	Mission^.XPick			:= WorkArea^[Mission^.PPick].X;// + (Layer^[WorkArea^[Mission^.PPick].Layer].X / 2); (* valorizzo la quota X di prelievo  *)
	Mission^.YPick			:= WorkArea^[Mission^.PPick].Y + (Layer^[WorkPickPointState^[Mission^.PPick].Code].YDim / 2); (* valorizzo la quota Y di prelievo *)
	Mission^.ZPick			:= WorkArea^[Mission^.PPick].Z; (* in questo modo LA LENTA va sempre fino a zero...mi fermo al raggiungimento dell'intervento dei tastatori *)
ELSE
	Errore.Code := ErrWAM_TipologiaMagazzinoFaldaNONRiconosciuta; (*Errore, Nell'impianto è stata impostata una tipologia di magazzino falde non prevista!!!*)
	RETURN;//EXIT;
END_IF
//IF WorkAreaState^[cwa].P = 0 THEN (* Se devo depositare la falda su una CASSA/CAVALLETTO *)
//(*******************************************************************************************************************************)	
//(********************************************* DEPOSITO FALDA SU CASSA/CAVALLETTO **********************************************)
//(*******************************************************************************************************************************)
TFWAM_CreaMissione_DepFaldaSuPallet(NPosInLavoro			:= Mission^.PPlace, //Numero Postazione di depositio
									Angolo_Destinazione 	:= Forming^[WorkAreaState^[Mission^.PPlace].F].PElement[WorkAreaState^[Mission^.PPlace].P].J, //Angolo di deposito dell'elemento
									PosizioneAttuale_X      := ModuleAX_X^.Ax^.Status.ActPosition, //Posizione attuale asse X
									TipologiaTraiettoria    := Forming^[WorkAreaState^[cwa].F].PElement[WorkAreaState^[cwa].P].Trajectory,
									
									Quota_PostX				:= WorkArea^[Mission^.PPlace].X, //Quota X Postazione
									Quota_PostY				:= WorkArea^[Mission^.PPlace].Y, //Quota Y Postazione
									Quota_PostZ				:= WorkArea^[Mission^.PPlace].Z, //Quota Z Postazione
									Quota_PostJ				:= WorkArea^[Mission^.PPlace].Rx, //Quota J Postazione
									
									Offset_Postazione_X 	:= WorkAreaOffset^[Mission^.PPlace].X, //Offset X Postazione
									Offset_Postazione_Y 	:= WorkAreaOffset^[Mission^.PPlace].Y, //Offset Y Postazione
									Offset_Postazione_Z 	:= WorkAreaOffset^[Mission^.PPlace].Z, //Offset Z Postazione
									Offset_Postazione_J 	:= WorkAreaOffset^[Mission^.PPlace].Rx, //Offset J Postazione
									
									Pallet_DimX				:= Forming^[WorkAreaState^[Mission^.PPlace].F].Pallet.XDim, //Dimensione X Pallet
									Pallet_DimY				:= Forming^[WorkAreaState^[Mission^.PPlace].F].Pallet.YDim, //Dimensione Y Pallet
									Pallet_DimZ				:= Forming^[WorkAreaState^[Mission^.PPlace].F].Pallet.ZDim, //Dimensione Z Pallet
									
									Offset_Pallet_X_0		:= Forming^[WorkAreaState^[Mission^.PPlace].F].Pallet.OFSDE_X0, //Offset X Pallet o Casse
									Offset_Pallet_Y_0		:= Forming^[WorkAreaState^[Mission^.PPlace].F].Pallet.OFSDE_Y0, //Offset Y Pallet o Casse 
									Offset_Pallet_Z_0		:= Forming^[WorkAreaState^[Mission^.PPlace].F].Pallet.OFSDE_Z0, //Offset Z Pallet o Casse + è grande + il deposito si distanzia dal supporto
									Offset_Pallet_J_0		:= Forming^[WorkAreaState^[Mission^.PPlace].F].Pallet.OFSDE_J0, //Offset J Pallet o Casse + è grande + la lastra sarà inclinata verso l'angolo crescente
									
									Offset_Pallet_X_90		:= Forming^[WorkAreaState^[Mission^.PPlace].F].Pallet.OFSDE_X90, //Offset X Pallet lato 0-90 
									Offset_Pallet_Y_90		:= Forming^[WorkAreaState^[Mission^.PPlace].F].Pallet.OFSDE_Y90, //Offset Y Pallet lato 0-90 + è grande + il deposito si distanzia dal supporto
									Offset_Pallet_Z_90		:= Forming^[WorkAreaState^[Mission^.PPlace].F].Pallet.OFSDE_Z90, //Offset Z Pallet lato 0-90 + è grande + il deposito si distanzia dal supporto
									Offset_Pallet_J_90		:= Forming^[WorkAreaState^[Mission^.PPlace].F].Pallet.OFSDE_J90, //Offset J Pallet lato 0-90 + è grande + la lastra sarà inclinata in fase di deposito
									
									Offset_Pallet_X_180		:= Forming^[WorkAreaState^[Mission^.PPlace].F].Pallet.OFSDE_X180, //Offset X Pallet lato 90-180
									Offset_Pallet_Y_180		:= Forming^[WorkAreaState^[Mission^.PPlace].F].Pallet.OFSDE_Y180, //Offset Y Pallet lato 90-180 + è grande + il deposito si distanzia dal supporto
									Offset_Pallet_Z_180		:= Forming^[WorkAreaState^[Mission^.PPlace].F].Pallet.OFSDE_Z180, //Offset Z Pallet lato 90-180 + è grande + il deposito si distanzia dal supporto
									Offset_Pallet_J_180		:= Forming^[WorkAreaState^[Mission^.PPlace].F].Pallet.OFSDE_J180, //Offset J Pallet lato 90-180 + è grande + la lastra sarà inclinata in fase di deposito
									
									Quota_FormaturaX 		:= Forming^[WorkAreaState^[Mission^.PPlace].F].PElement[WorkAreaState^[Mission^.PPlace].P].X, //Quota Deposito X da Formatura
									Quota_FormaturaY 		:= Forming^[WorkAreaState^[Mission^.PPlace].F].PElement[WorkAreaState^[Mission^.PPlace].P].Y, //Quota Deposito Y da Formatura
									Quota_FormaturaZ 		:= Forming^[WorkAreaState^[Mission^.PPlace].F].PElement[WorkAreaState^[Mission^.PPlace].P].Z, //Quota Deposito Z da Formatura
									Quota_FormaturaJ 		:= Forming^[WorkAreaState^[Mission^.PPlace].F].PElement[WorkAreaState^[Mission^.PPlace].P].J, //Quota Deposito Z da Formatura
									
									Distanza_ApproccioFormaturaX 		:= Forming^[WorkAreaState^[Mission^.PPlace].F].PElement[WorkAreaState^[Mission^.PPlace].P].AX, //Distanza Deposito X da Formatura
									Distanza_ApproccioFormaturaY 		:= Forming^[WorkAreaState^[Mission^.PPlace].F].PElement[WorkAreaState^[Mission^.PPlace].P].AY, //Distanza Deposito Y da Formatura
									Distanza_ApproccioFormaturaZ 		:= Forming^[WorkAreaState^[Mission^.PPlace].F].PElement[WorkAreaState^[Mission^.PPlace].P].AZ, //Distanza Deposito Z da Formatura
									Distanza_ApproccioFormaturaJ 		:= Forming^[WorkAreaState^[Mission^.PPlace].F].PElement[WorkAreaState^[Mission^.PPlace].P].AJ, //Distanza Deposito Z da Formatura
									
									Quota_DestX 			=> Mission^.XPlace, //Quota DESTINAZIONE X
									Quota_DestY 			=> Mission^.YPlace, //Quota DESTINAZIONE Y
									Quota_DestZ 			=> Mission^.ZPlace, //Quota DESTINAZIONE Z
									Quota_DestJ 			=> Mission^.JPlace, //Quota DESTINAZIONE J	
									
									Quota_ApproccioDestX 	=> Mission^.XPlaceApproach, //Quota APPROCCIO di DESTINAZIONE X
									Quota_ApproccioDestY 	=> Mission^.YPlaceApproach, //Quota APPROCCIO di DESTINAZIONE Y
									Quota_ApproccioDestZ 	=> Mission^.ZPlaceApproach, //Quota APPROCCIO di DESTINAZIONE Z
									Quota_ApproccioDestJ 	=> Mission^.JPlaceApproach);//Quota APPROCCIO di DESTINAZIONE J	
	IF TFWAM_CreaMissione_DepFaldaSuPallet.Errore.Code > 0 THEN
		Errore := TFWAM_CreaMissione_DepFaldaSuPallet.Errore;
		RETURN;//EXIT;
	END_IF
	CASE Forming^[WorkAreaState^[Mission^.PPlace].F].Pallet.Tipologia OF
		CAVALLETTO :
			IF Forming^[WorkAreaState^[Mission^.PPlace].F].PElement[WorkAreaState^[Mission^.PPlace].P].J > 90 THEN (* Se devo depositare la falda su CAVALLETTO lato 180°*)	
				Mission^.XDim			:= Layer^[Forming^[WorkAreaState^[cwa].F].PElement[WorkAreaState^[Mission^.PPlace].P].TypologyCode].XDim ;
				Mission^.YDim			:= Layer^[Forming^[WorkAreaState^[cwa].F].PElement[WorkAreaState^[Mission^.PPlace].P].TypologyCode].YDim;
				Mission^.ZDim			:= Layer^[Forming^[WorkAreaState^[cwa].F].PElement[WorkAreaState^[Mission^.PPlace].P].TypologyCode].ZDim;
			ELSIF Forming^[WorkAreaState^[Mission^.PPlace].F].PElement[WorkAreaState^[Mission^.PPlace].P].J < 90 THEN (* Se devo depositare la falda su CAVALLETTO lato 0°*)		
				Mission^.XDim			:= Layer^[Forming^[WorkAreaState^[cwa].F].PElement[WorkAreaState^[Mission^.PPlace].P].TypologyCode].XDim ;
				Mission^.YDim			:= Layer^[Forming^[WorkAreaState^[cwa].F].PElement[WorkAreaState^[Mission^.PPlace].P].TypologyCode].YDim;
				Mission^.ZDim			:= Layer^[Forming^[WorkAreaState^[cwa].F].PElement[WorkAreaState^[Mission^.PPlace].P].TypologyCode].ZDim;
			END_IF
			WorkAreaManager^.State := WAMANAGER_CICLO_PRELIEVO_FALDA_RUN;	(* Set Stato del WorkAreaManager *)
			RestoreCWA^ := TRUE;
			PreviousPWA^ := pwa;
			RETURN;//EXIT;
		CASSA_STANDARD :
			Mission^.XDim			:= Layer^[Forming^[WorkAreaState^[cwa].F].PElement[WorkAreaState^[Mission^.PPlace].P].TypologyCode].XDim ;
			Mission^.YDim			:= Layer^[Forming^[WorkAreaState^[cwa].F].PElement[WorkAreaState^[Mission^.PPlace].P].TypologyCode].YDim;
			Mission^.ZDim			:= Layer^[Forming^[WorkAreaState^[cwa].F].PElement[WorkAreaState^[Mission^.PPlace].P].TypologyCode].ZDim;
			WorkAreaManager^.State := WAMANAGER_CICLO_PRELIEVO_FALDA_RUN;	(* Set Stato del WorkAreaManager *)
			RestoreCWA^ := TRUE;
			PreviousPWA^ := pwa;
			RETURN;//EXIT;
	ELSE
		Errore.Code := ErrWAM_TipologiaPalletNONRiconosciuta; 		(* Genero un errore che mi indica che la tipologia di "Pallet/Cassa/Cavallina" non è riconosciuto *)
		RETURN;//EXIT;		
	END_CASE
END_ACTION

ACTION LASTRA_PP_INIT:
(* Reset della memoria utilizzata per forzare il ciclo di riposo in ciclo di prelievo pacco *)
ForzaPrelievoPaccoDuranteCicloDiRiposo := FALSE;			
(* Definisco che la WORKAREA è positiva -> Default per lastre! *)
Mission^.PPick 	:= ppick;								   			// Assegno il numero del Punto di prelievo
Mission^.TPick 	:= TPICK_LASTRA;									// Assegno il tipo di Prelievo
Mission^.PPlace := cwa;									   			// Assegno il numero della piazzola di deposito
Mission^.XDim 	:= WorkPickPointState^[Mission^.PPick].Element.XDim ; 	// Assegno la dimensione X del pacco presente nel punto di prelievo designato
Mission^.YDim 	:= WorkPickPointState^[Mission^.PPick].Element.YDim; 	// Assegno la dimensione X del pacco presente nel punto di prelievo designato
Mission^.ZDim 	:= WorkPickPointState^[Mission^.PPick].Element.ZDim; 	// Assegno la dimensione X del pacco presente nel punto di prelievo designato

(* Calcolo Delle quote di Prelievo *)
XPick := TFPalletizer_CalcolaCoordinataPrelievo_PickPoint(WorkPickPoint,WorkPickPointState,WorkPickPointOffset,Mission^.PPick,'X');		
YPick := TFPalletizer_CalcolaCoordinataPrelievo_PickPoint(WorkPickPoint,WorkPickPointState,WorkPickPointOffset,Mission^.PPick,'Y');
ZPick := TFPalletizer_CalcolaCoordinataPrelievo_PickPoint(WorkPickPoint,WorkPickPointState,WorkPickPointOffset,Mission^.PPick,'Z');
JPick := TFPalletizer_CalcolaCoordinataPrelievo_PickPoint(WorkPickPoint,WorkPickPointState,WorkPickPointOffset,Mission^.PPick,'J');	

(* Assegnazione quote alla Missione *)
Mission^.XPick			:= XPick;
Mission^.YPick			:= YPick;
Mission^.ZPick			:= ZPick;
Mission^.JPick			:= JPick;

Mission^.XPickApproach	:= XPick;							
Mission^.YPickApproach	:= YPick;	  
Mission^.ZPickApproach	:= ZPick + PickPlaceParameters^.ZPickApproach;//Quota prelievo + offset approccio... in mod da fare la lenta ottimizzata
Mission^.JPickApproach	:= JPick;	
	
(* Set delle variabili per andare al punto di riposo *)
X_Riposo	:= XPick;
Y_Riposo	:= YPick;
J_Riposo	:= JPick;
Z_Riposo	:= QuotaFuoriIngombro_Z_AVUOTO;		

IF WorkAreaState^[Mission^.PPlace].Apprendimento.Z.Lato90.Stato <> APPRENDIMENTO_ESEGUITO THEN
	IF WorkareaState^[Mission^.PPlace].TransportState.Supporto.Tipologia = e_Tipo_Pallet.CASSA_STANDARD THEN 
		WorkAreaState^[Mission^.PPlace].Apprendimento.Z.Lato90.QuotaStart 	:= 950;
	ELSE
		WorkAreaState^[Mission^.PPlace].Apprendimento.Z.Lato90.QuotaStart 	:= 950;
	END_IF
END_IF
//Disabilito apprendimento in deposito se disabilitato
IF NOT HMI_AbilitaDepositoPaccoOrrizzontaleConTasteggio THEN
	WorkAreaState^[Mission^.PPlace].Apprendimento.Z.Lato90.Stato := APPRENDIMENTO_DISABILITATO;
END_IF
(* Calcolo gli ingombri della pinza nelle varie direzioni *)
IF Forming^[WorkAreaState^[Mission^.PPlace].F].PElement[WorkAreaState^[Mission^.PPlace].P].J <= 87 THEN
	LatoDeposito := 0;
ELSIF Forming^[WorkAreaState^[Mission^.PPlace].F].PElement[WorkAreaState^[Mission^.PPlace].P].J >= 93 THEN
	LatoDeposito := 180;
END_IF
							
TFCalcoliIngombroPinza(Mission := Mission,
					WorkAreaManager := WorkAreaManager,
					WorkAreaState := ADR(WorkAreaState),
					ModuleAX_J := ModuleAX_J,
					AngoloRotazioneDestinazionePinza:= Forming^[WorkAreaState^[Mission^.PPlace].F].PElement[WorkAreaState^[Mission^.PPlace].P].J,
					IngombroX_Pos 				:= ADR(IngombroX_Pos),
					IngombroY_Pos 				:= ADR(IngombroY_Pos),
					IngombroX_Neg 				:= ADR(IngombroX_Neg),
					IngombroY_Neg 				:= ADR(IngombroY_Neg),
					IngombroZ_Pos 				:= ADR(IngombroZ_Pos),
					IngombroZ_Neg 				:= ADR(IngombroZ_Neg),
					IngombroY_Tot 				:= ADR(IngombroY_Tot),
					IngombroDestinazioneX_Pos 	:= ADR(IngombroDestinazioneX_Pos),
					IngombroDestinazioneY_Pos 	:= ADR(IngombroDestinazioneY_Pos),
					IngombroDestinazioneX_Neg 	:= ADR(IngombroDestinazioneX_Neg),
					IngombroDestinazioneY_Neg 	:= ADR(IngombroDestinazioneY_Neg),
					IngombroDestinazioneZ_Pos 	:= ADR(IngombroDestinazioneZ_Pos),
					IngombroDestinazioneZ_Neg 	:= ADR(IngombroDestinazioneZ_Neg),
					IngombroMaxX_Pos 			:= ADR(IngombroMaxX_Pos),
					IngombroMaxY_Pos 			:= ADR(IngombroMaxY_Pos),
					IngombroMaxX_Neg 			:= ADR(IngombroMaxX_Neg),
					IngombroMaxY_Neg 			:= ADR(IngombroMaxY_Neg),
					IngombroMaxZ_Pos 			:= ADR(IngombroMaxZ_Pos),
					IngombroMaxZ_Neg 			:= ADR(IngombroMaxZ_Neg),
					IngombroY_Pos_0  			:= ADR(IngombroY_Pos_0),		 		
					IngombroY_Neg_180 			:= ADR(IngombroY_Neg_180),
					IngombroY_Neg_0 			:= ADR(IngombroY_Neg_0),	
					IngombroY_Pos_180 			:= ADR(IngombroY_Pos_180),
					ScostamentoVerticalePuntoCentrale := ADR(ScostamentoVerticalePuntoCentrale));

(* Valorizzazione quote di deposito Ciclo Lastra *)
TFWAM_CreaMissione_DepLastraDaPP(NPosInLavoro			    := Mission^.PPlace, //Numero Postazione di depositio
									Angolo_Destinazione 	:= Forming^[WorkAreaState^[Mission^.PPlace].F].PElement[WorkAreaState^[Mission^.PPlace].P].J, //Angolo di deposito dell'elemento
									PosizioneAttuale_X      := ModuleAX_X^.Ax^.Status.ActPosition, //Posizione attuale asse X
									TipologiaTraiettoria    := TRAIETTORIA_CON_APPROCCIO,//Forming^[WorkAreaState^[cwa].F].PElement[WorkAreaState^[cwa].P].Trajectory,
									Apprendimento			:= WorkAreaState^[Mission^.PPlace].Apprendimento,
									CicloDiPrelievo         := FALSE,
									HmaxElemento			:= WorkAreaState^[Mission^.PPlace].TransportState.Supporto.HMAX,
									Offset_Apprendimento_X 	:= 0,//OffsetApprendimento.Lastra.X, //Offset X Postazione,
									Offset_Apprendimento_Y 	:= OffsetApprendimento.Lastra.Y, //Offset Y Postazione
									Offset_Apprendimento_Z 	:= OffsetApprendimento.Lastra.Z, //Offset Z Postazione
									Offset_Apprendimento_J 	:= 0,//OffsetApprendimento.Lastra.J, //Offset J Postazione

									Quota_PostX				:= WorkArea^[Mission^.PPlace].X, //Quota X Postazione
									Quota_PostY				:= WorkArea^[Mission^.PPlace].Y, //Quota Y Postazione
									Quota_PostZ				:= WorkArea^[Mission^.PPlace].Z, //Quota Z Postazione
									Quota_PostJ				:= WorkArea^[Mission^.PPlace].Rx, //Quota J Postazione
									
									Offset_Postazione_X 	:= WorkAreaOffset^[Mission^.PPlace].X, //Offset X Postazione
									Offset_Postazione_Y 	:= WorkAreaOffset^[Mission^.PPlace].Y, //Offset Y Postazione
									Offset_Postazione_Z 	:= WorkAreaOffset^[Mission^.PPlace].Z, //Offset Z Postazione
									Offset_Postazione_J 	:= WorkAreaOffset^[Mission^.PPlace].Rx, //Offset J Postazione
									
									Pallet_DimX				:= WorkAreaState^[Mission^.PPlace].Supporto.XDim, //Dimensione X Pallet
									Pallet_DimY				:= WorkAreaState^[Mission^.PPlace].Supporto.YDim, //Dimensione Y Pallet
									Pallet_DimZ				:= WorkAreaState^[Mission^.PPlace].Supporto.ZDim, //Dimensione Z Pallet
									
									Quota_FormaturaX 		:= Forming^[WorkAreaState^[Mission^.PPlace].F].PElement[WorkAreaState^[Mission^.PPlace].P].X, //Quota Deposito X da Formatura
									Quota_FormaturaY 		:= ABS(Forming^[WorkAreaState^[Mission^.PPlace].F].PElement[WorkAreaState^[Mission^.PPlace].P].Y), //Quota Deposito Y da Formatura
									Quota_FormaturaZ 		:= Forming^[WorkAreaState^[Mission^.PPlace].F].PElement[WorkAreaState^[Mission^.PPlace].P].Z, //Quota Deposito Z da Formatura
									Quota_FormaturaJ 		:= Forming^[WorkAreaState^[Mission^.PPlace].F].PElement[WorkAreaState^[Mission^.PPlace].P].J, //Quota Deposito Z da Formatura
									
									Distanza_ApproccioFormaturaX 		:= Forming^[WorkAreaState^[Mission^.PPlace].F].PElement[WorkAreaState^[Mission^.PPlace].P].AX, //Quota Deposito X da Formatura
									Distanza_ApproccioFormaturaY 		:= PickPlaceParameters^.YPlaceApproach, 
									Distanza_ApproccioFormaturaZ 		:= PickPlaceParameters^.ZPlaceApproach,
									Distanza_ApproccioFormaturaJ 		:= Forming^[WorkAreaState^[Mission^.PPlace].F].PElement[WorkAreaState^[Mission^.PPlace].P].AJ, //Quota Deposito Z da Formatura
									
									Quota_DestX 			=> Mission^.XPlace, //Quota DESTINAZIONE X
									Quota_DestY 			=> Mission^.YPlace, //Quota DESTINAZIONE Y
									Quota_DestZ 			=> Mission^.ZPlace, //Quota DESTINAZIONE Z
									Quota_DestJ 			=> Mission^.JPlace, //Quota DESTINAZIONE J	
									
									Quota_ApproccioDestX 	=> Mission^.XPlaceApproach, //Quota APPROCCIO di DESTINAZIONE X
									Quota_ApproccioDestY 	=> Mission^.YPlaceApproach, //Quota APPROCCIO di DESTINAZIONE Y
									Quota_ApproccioDestZ 	=> Mission^.ZPlaceApproach, //Quota APPROCCIO di DESTINAZIONE Z
									Quota_ApproccioDestJ 	=> Mission^.JPlaceApproach);//Quota APPROCCIO di DESTINAZIONE J	

IF TFWAM_CreaMissione_DepLastraDaPP.Errore.Code > 0 THEN
	Errore := TFWAM_CreaMissione_DepLastraDaPP.Errore;
	RETURN;//EXIT;
ELSE
	RestoreCWA^ := TRUE;
	PreviousPWA^ := pwa;
	WorkAreaManager^.State 	:= WAMANAGER_CICLO_PRELIEVO_LASTRA_PP_RUN;
END_IF
(* Setto l'uscita che mi determina il deposito del primo pacco in lenta *)
IF WorkAreaState^[Mission^.PPlace].Slow = 1 THEN
	DepositoPaccoInLenta := TRUE;
END_IF
END_ACTION

ACTION LASTRA_WA_INIT:
Mission^.PPlace	:= cwa; (* valorizzo il punto di deposito *)
(* Aggiorno la struttura delle Lastre in missione *)
Mission^.Slab := WorkAreaState^[Mission^.PPick].Slab[WorkAreaState^[cwa].P];

NLastraDaPrelevare := WorkAreaState^[Mission^.PPick].P-1;
IF NLastraDaPrelevare >= 1 THEN
	NLastraDaPrelevare := 1 ;// añadido para probar
ELSE
	Errore.Code := ErrWA_NumPezzInPrelErrato;
	RETURN;
END_IF


				
Mission^.TPick 	:= TPICK_LASTRA;	// Assegno il tipo di Prelievo
Mission^.XDim 	:= Forming^[WorkAreaState^[Mission^.PPlace].F].PElement[NLastraDaPrelevare].XDim;// WorkAreaState^[Mission^.PPick].Slab[NLastraDaPrelevare].XDim;	// Assegno la dimensione X del pacco presente nel punto di prelievo designato
Mission^.YDim 	:= Forming^[WorkAreaState^[Mission^.PPlace].F].PElement[NLastraDaPrelevare].YDim;//WorkAreaState^[Mission^.PPick].Slab[NLastraDaPrelevare].YDim;	// Assegno la dimensione Y del pacco presente nel punto di prelievo designato
Mission^.ZDim 	:= Forming^[WorkAreaState^[Mission^.PPlace].F].PElement[NLastraDaPrelevare].ZDim;//WorkAreaState^[Mission^.PPick].Slab[NLastraDaPrelevare].ZDim; 	// Assegno la dimensione Z del pacco presente nel punto di prelievo designato
ppick := Mission^.PPick;

IF Mission^.XDim <=0	OR Mission^.YDim <= 0 THEN
	Errore.Code := ErrEsMisionSinDimesionPieza;
	RETURN;
END_IF
(* Valorizzazione del lato di prelievo nel caso di prelievo su cavallina *)
IF WorkareaState^[Mission^.PPick].Supporto.Tipologia = e_Tipo_Pallet.BUNDLE THEN //Se ho in prelievo il supporto di tipo bundle
	IF ppickOld <> Mission^.PPick THEN 	//Ad ogni cambio di postazione setto il valore del lato iniziale a 0
		TFClearApprendimento(ADR(WorkAreaState^[Mission^.PPick].Apprendimento));//Pulisco la struttura dell'apprendimento
		LatoPrelievo := 180;				//Vado a prelevare sul lato 180	
		TFWAM_CreaMissione_PrelLastraDaWA.Quota_FormaturaJ := 180; //Assegno la quota di 0° per il prelievo, in questo modo la pinza parte a fare il tasteggio in questa posizione					
		IF LatoPrelievo = 0 THEN
		(* Apprendimento lungo X *)
			WorkAreaState^[Mission^.PPick].Apprendimento.X.Lato0.Stato		:= APPRENDIMENTO_DISABILITATO;
			WorkAreaState^[Mission^.PPick].Apprendimento.Y.Lato0.Stato		:= APPRENDIMENTO_DA_ESEGUIRE;
		ELSIF LatoPrelievo = 180 THEN
			WorkAreaState^[Mission^.PPick].Apprendimento.X.Lato180.Stato	:= APPRENDIMENTO_DISABILITATO;
			WorkAreaState^[Mission^.PPick].Apprendimento.Y.Lato180.Stato	:= APPRENDIMENTO_DA_ESEGUIRE;
		END_IF
	ELSE
		LatoPrelievo := 180;				//Vado a prelevare sul lato 180	
		TFWAM_CreaMissione_PrelLastraDaWA.Quota_FormaturaJ := 180; //Assegno la quota di 0° per il prelievo, in questo modo la pinza parte a fare il tasteggio in questa posizione					
		IF LatoPrelievo = 0 THEN
		(* Apprendimento lungo X *)
			WorkAreaState^[Mission^.PPick].Apprendimento.X.Lato0.Stato		:= APPRENDIMENTO_DISABILITATO;
			IF WorkAreaState^[Mission^.PPick].Apprendimento.Y.Lato0.Stato <> APPRENDIMENTO_ESEGUITO THEN
				WorkAreaState^[Mission^.PPick].Apprendimento.Y.Lato0.Stato		:= APPRENDIMENTO_DA_ESEGUIRE;
			END_IF
		ELSIF LatoPrelievo = 180 THEN
			WorkAreaState^[Mission^.PPick].Apprendimento.X.Lato180.Stato	:= APPRENDIMENTO_DISABILITATO;
			IF WorkAreaState^[Mission^.PPick].Apprendimento.Y.Lato180.Stato <> APPRENDIMENTO_ESEGUITO THEN
				WorkAreaState^[Mission^.PPick].Apprendimento.Y.Lato180.Stato	:= APPRENDIMENTO_DA_ESEGUIRE;
			END_IF
		END_IF
	END_IF
ELSIF WorkareaState^[Mission^.PPick].Supporto.Tipologia = e_Tipo_Pallet.CAVALLETTO THEN //Se ho in prelievo il supporto di tipo cavalletto
	
	AguloDeRecogida := FunLadoTrabajoCaballete(Piezas_LadoA := 
						HMI_NumeroPezziPresentiCavallete[Mission^.PPick].HMI_NumeroPezziPresentiPostazione_A_Cavaleto , 
							Piezas_Ladob := HMI_NumeroPezziPresentiCavallete[Mission^.PPick].HMI_NumeroPezziPresentiPostazione_B_Cavaleto ,
								Recoger := TRUE ,dejar := FALSE ,GestionLadoTrabajo := WorkareaState^[Mission^.PPick].Supporto.TipoTrabajoLado_Cavallete ,
									GestionDescargaCaballete := ADR(GestionDescargaCaballete) 	);
	LatoPrelievo := AguloDeRecogida ;
	IF FALSE THEN 
			IF FormaturaAFRAMERT[WorkAreaState^[Mission^.PPlace].F].PElement[WorkAreaState^[Mission^.PPick].P-1].J > 90 THEN
				LatoPrelievo := 180;
			
			ELSIF FormaturaAFRAMERT[WorkAreaState^[Mission^.PPlace].F].PElement[WorkAreaState^[Mission^.PPick].P-1].J  < 90 THEN
				LatoPrelievo := 0;
			END_IF	
	END_IF
	
	IF ppickOld <> Mission^.PPick THEN 	//Ad ogni cambio di postazione setto il valore del lato iniziale a 0
		TFClearApprendimento(ADR(WorkAreaState^[Mission^.PPick].Apprendimento));//Pulisco la struttura dell'apprendimento
		TFWAM_CreaMissione_PrelLastraDaWA.Quota_FormaturaJ := 180; //Assegno la quota di 0° per il prelievo, in questo modo la pinza parte a fare il tasteggio in questa posizione					
		WorkAreaState^[Mission^.PPick].Apprendimento.X.Lato0.Stato		:= APPRENDIMENTO_DISABILITATO;
		WorkAreaState^[Mission^.PPick].Apprendimento.Y.Lato0.Stato		:= APPRENDIMENTO_DA_ESEGUIRE;
		WorkAreaState^[Mission^.PPick].Apprendimento.X.Lato180.Stato	:= APPRENDIMENTO_DISABILITATO;
		WorkAreaState^[Mission^.PPick].Apprendimento.Y.Lato180.Stato	:= APPRENDIMENTO_DA_ESEGUIRE;
	ELSE
		TFWAM_CreaMissione_PrelLastraDaWA.Quota_FormaturaJ := 180; //Assegno la quota di 0° per il prelievo, in questo modo la pinza parte a fare il tasteggio in questa posizione					
		IF LatoPrelievo = 0 THEN
		(* Apprendimento lungo X *)
			WorkAreaState^[Mission^.PPick].Apprendimento.X.Lato0.Stato		:= APPRENDIMENTO_DISABILITATO;
			IF WorkAreaState^[Mission^.PPick].Apprendimento.Y.Lato0.Stato <> APPRENDIMENTO_ESEGUITO THEN
				WorkAreaState^[Mission^.PPick].Apprendimento.Y.Lato0.Stato		:= APPRENDIMENTO_DA_ESEGUIRE;
				//WorkAreaState^[Mission^.PPick].Apprendimento.Y.Lato0.QuotaStart	:= 1000;
			END_IF
		ELSIF LatoPrelievo = 180 THEN
			WorkAreaState^[Mission^.PPick].Apprendimento.X.Lato180.Stato	:= APPRENDIMENTO_DISABILITATO;
			IF WorkAreaState^[Mission^.PPick].Apprendimento.Y.Lato180.Stato <> APPRENDIMENTO_ESEGUITO THEN
				WorkAreaState^[Mission^.PPick].Apprendimento.Y.Lato180.Stato	:= APPRENDIMENTO_DA_ESEGUIRE;
				//WorkAreaState^[Mission^.PPick].Apprendimento.Y.Lato180.QuotaStart	:= 1000;
			END_IF
		END_IF
	END_IF
ELSIF WorkareaState^[Mission^.PPick].Supporto.Tipologia <> e_Tipo_Pallet.CAVALLETTO AND WorkareaState^[Mission^.PPick].Supporto.Tipologia <> e_Tipo_Pallet.BUNDLE THEN //Se NON ho in prelievo il supporto di tipo cavalletto
	LatoPrelievo := 90; //Setto il lato di prelievo = 90
	IF ppickOld <> ppick THEN 	//Ad ogni cambio di postazione setto il valore del lato iniziale a 0
		TFClearApprendimento(ADR(WorkAreaState^[Mission^.PPick].Apprendimento));//Pulisco la struttura dell'apprendimento
	END_IF
	TFWAM_CreaMissione_PrelLastraDaWA.Quota_FormaturaJ := 90;//Assegno la quota di 90° per il prelievo, in questo modo la pinza preleverà in orizzontale
	IF WorkAreaState^[Mission^.PPick].Apprendimento.Z.Lato90.Stato <> APPRENDIMENTO_ESEGUITO THEN
		WorkAreaState^[Mission^.PPick].Apprendimento.Z.Lato90.Stato := APPRENDIMENTO_DA_ESEGUIRE;
		IF WorkareaState^[Mission^.PPick].Supporto.Tipologia = e_Tipo_Pallet.CASSA_STANDARD THEN 
			WorkAreaState^[Mission^.PPick].Apprendimento.Z.Lato90.QuotaStart 	:= 700;
		ELSE
			WorkAreaState^[Mission^.PPick].Apprendimento.Z.Lato90.QuotaStart 	:= 700;
		END_IF
	END_IF
END_IF

//Disabilito apprendimento in deposito se disabilitato
IF NOT HMI_AbilitaDepositoPaccoOrrizzontaleConTasteggio AND FALSE THEN
	WorkAreaState^[Mission^.PPick].Apprendimento.Z.Lato90.Stato := APPRENDIMENTO_DISABILITATO;	
END_IF

(* Memorizzo l'ultima postazione in cui è stato effettuato il prelievo *)
UltimaPostazioneInPrelievo := Mission^.PPick;
ppickOld := Mission^.PPick;

IF HabilitacionFormacionNueva THEN
	FormaturaBundleRT[WorkAreaProductionList^[Mission^.PPlace].NumeroListaAssociata] := FormaturaWa[Mission^.PPick];
	FormaturaAFRAMERT[WorkAreaProductionList^[Mission^.PPlace].NumeroListaAssociata] := FormaturaWa[Mission^.PPick];
	;
END_IF


//Z prelievo a seconda della tipologia 
IF WorkareaState^[Mission^.PPick].Supporto.Tipologia = e_Tipo_Pallet.BUNDLE THEN //SE PRELIEVO SU BUNDLE O CASSA
	IF LatoPrelievo = 180 THEN
		AngoloPrelievo 					:= 180-2;
		AltezzaCentroLastraInclinata 	:=  	ABS((Mission^.YDim/2) * COS(DEG_TO_RAD(AngoloPrelievo)));
		QuotaLastraYRealTimePrelievo 			:= FormaturaBundleRT[WorkAreaProductionList^[Mission^.PPlace].NumeroListaAssociata].PElement[WorkAreaState^[Mission^.PPick].P-1].Y;
		QuotaLastraZRealTimePrelievo 			:= FormaturaBundleRT[WorkAreaProductionList^[Mission^.PPlace].NumeroListaAssociata].PElement[WorkAreaState^[Mission^.PPick].P-1].Z (*+  (*Dimensioni_Pinza.DimTraveVerticale / 2*) CuotaOffSetZRecogidaBundel *);
	ELSIF LatoPrelievo = 0 THEN
		AngoloPrelievo 							:= 2;
		AltezzaCentroLastraInclinata 			:=  ABS((Mission^.YDim/2) * COS(DEG_TO_RAD(AngoloPrelievo)));
		IF TRUE THEN 
			QuotaLastraYRealTimePrelievo 			:= FormaturaBundleRT[WorkAreaProductionList^[Mission^.PPlace].NumeroListaAssociata].PElement[WorkAreaState^[Mission^.PPick].P_Cava.HMI_NumeroPezziPresentiPostazione_A_Cavaleto-1].CooCavallete.LadoA.CoordenadaFinale_Y;
			QuotaLastraZRealTimePrelievo 			:= FormaturaBundleRT[WorkAreaProductionList^[Mission^.PPlace].NumeroListaAssociata].PElement[WorkAreaState^[Mission^.PPick].P_Cava.HMI_NumeroPezziPresentiPostazione_A_Cavaleto-1].CooCavallete.LadoA.CoordenadaFinale_Z;(*+  (*Dimensioni_Pinza.DimTraveVerticale / 2*) CuotaOffSetZRecogidaBundel *);
		ELSE
			QuotaLastraYRealTimePrelievo 			:= FormaturaBundleRT[WorkAreaProductionList^[Mission^.PPlace].NumeroListaAssociata].PElement[WorkAreaState^[Mission^.PPick].P-1].Y;
			QuotaLastraZRealTimePrelievo 			:= FormaturaBundleRT[WorkAreaProductionList^[Mission^.PPlace].NumeroListaAssociata].PElement[WorkAreaState^[Mission^.PPick].P-1].Z (*+ (*Dimensioni_Pinza.DimTraveVerticale / 2*) CuotaOffSetZRecogidaBundel*) ;		
			
		END_IF
		
	ELSE
		AngoloPrelievo := 90;
		AltezzaCentroLastraInclinata := 0;
		QuotaLastraZRealTimePrelievo := 0;
		QuotaLastraYRealTimePrelievo := 0;
	END_IF
ELSIF WorkareaState^[Mission^.PPick].Supporto.Tipologia = e_Tipo_Pallet.CAVALLETTO THEN
	IF LatoPrelievo = 180 THEN
		AngoloPrelievo 					:= 180-2;
		AltezzaCentroLastraInclinata 	:= ABS((Mission^.YDim/2) * COS(DEG_TO_RAD(AngoloPrelievo)));
		IF TRUE THEN
			QuotaLastraYRealTimePrelievo 			:= FormaturaAFRAMERT[WorkAreaProductionList^[Mission^.PPlace].NumeroListaAssociata].PElement[WorkAreaState^[Mission^.PPick].P_Cava.HMI_NumeroPezziPresentiPostazione_B_Cavaleto-1].CooCavallete.LadoB.CoordenadaFinale_Y;
			QuotaLastraZRealTimePrelievo 			:= FormaturaAFRAMERT[WorkAreaProductionList^[Mission^.PPlace].NumeroListaAssociata].PElement[WorkAreaState^[Mission^.PPick].P_Cava.HMI_NumeroPezziPresentiPostazione_B_Cavaleto-1].CooCavallete.LadoB.CoordenadaFinale_Z;(*+  (*Dimensioni_Pinza.DimTraveVerticale / 2*) CuotaOffSetZRecogidaBundel *);
		ELSE
 			QuotaLastraYRealTimePrelievo 			:= FormaturaAFRAMERT[WorkAreaProductionList^[Mission^.PPlace].NumeroListaAssociata].PElement[WorkAreaState^[Mission^.PPick].P-1].Y;
			QuotaLastraZRealTimePrelievo 			:= FormaturaAFRAMERT[WorkAreaProductionList^[Mission^.PPlace].NumeroListaAssociata].PElement[WorkAreaState^[Mission^.PPick].P-1].Z + (*Dimensioni_Pinza.DimTraveVerticale / 2*) CuotaOffSetZRecogidaCaballete;
		END_IF
	ELSIF LatoPrelievo = 0 THEN
		AngoloPrelievo 					:= 3;
		AltezzaCentroLastraInclinata 	:= ABS((Mission^.YDim/2) * COS(DEG_TO_RAD(AngoloPrelievo)));
		IF TRUE THEN 
			QuotaLastraYRealTimePrelievo 			:= FormaturaAFRAMERT[WorkAreaProductionList^[Mission^.PPlace].NumeroListaAssociata].PElement[WorkAreaState^[Mission^.PPick].P_Cava.HMI_NumeroPezziPresentiPostazione_A_Cavaleto-1].CooCavallete.LadoA.CoordenadaFinale_Y;
			QuotaLastraZRealTimePrelievo 			:= FormaturaAFRAMERT[WorkAreaProductionList^[Mission^.PPlace].NumeroListaAssociata].PElement[WorkAreaState^[Mission^.PPick].P_Cava.HMI_NumeroPezziPresentiPostazione_A_Cavaleto-1].CooCavallete.LadoA.CoordenadaFinale_Z;(*+  (*Dimensioni_Pinza.DimTraveVerticale / 2*) CuotaOffSetZRecogidaBundel *);
		ELSE
			QuotaLastraYRealTimePrelievo 			:= FormaturaAFRAMERT[WorkAreaProductionList^[Mission^.PPlace].NumeroListaAssociata].PElement[WorkAreaState^[Mission^.PPick].P-1].Y;
			QuotaLastraZRealTimePrelievo 			:= FormaturaAFRAMERT[WorkAreaProductionList^[Mission^.PPlace].NumeroListaAssociata].PElement[WorkAreaState^[Mission^.PPick].P-1].Z (*+ (*Dimensioni_Pinza.DimTraveVerticale / 2*) CuotaOffSetZRecogidaCaballete *);
		END_IF
	ELSE
		AngoloPrelievo := 90;
		AltezzaCentroLastraInclinata := 0;
		QuotaLastraZRealTimePrelievo := 0;
		QuotaLastraYRealTimePrelievo := 0;
	END_IF
ELSE
	IF LatoPrelievo = 90 THEN		
		AngoloPrelievo := 90;
		AltezzaCentroLastraInclinata := 0;
		QuotaLastraZRealTimePrelievo := 0;
		QuotaLastraYRealTimePrelievo := 0;
	ELSE
		Errore.Code := ErrWA_SupportoInPrelivoNonPrevisto;
	END_IF
END_IF

//CALCOLO INGOMBRI PINZA						

;
//OffSetZRecogidaEnAngulo				:=  -20 ;					
//ScostamentoVerticalePuntoCentrale := ABS(Dimensioni_Pinza.Spessore * COS(deg_to_rad(-90+AngoloPrelievo))-Dimensioni_Pinza.Spessore);

// Calculo Del Ingombro Pinza Mision Recogida lastra
TFCalcoliIngombroPinza(Mission := Mission,
						WorkAreaManager := WorkAreaManager,
						WorkAreaState := ADR(WorkAreaState),
						ModuleAX_J := ModuleAX_J,
						AngoloRotazioneDestinazionePinza:= LatoPrelievo,//Forming^[WorkAreaState^[Mission^.PPlace].F].PElement[WorkAreaState^[Mission^.PPlace].P].J+2,
						IngombroX_Pos 				:= ADR(IngombroX_Pos),
						IngombroY_Pos 				:= ADR(IngombroY_Pos),
						IngombroX_Neg 				:= ADR(IngombroX_Neg),
						IngombroY_Neg 				:= ADR(IngombroY_Neg),
						IngombroZ_Pos 				:= ADR(IngombroZ_Pos),
						IngombroZ_Neg 				:= ADR(IngombroZ_Neg),
						IngombroY_Tot 				:= ADR(IngombroY_Tot),
						IngombroDestinazioneX_Pos 	:= ADR(IngombroDestinazioneX_Pos),
						IngombroDestinazioneY_Pos 	:= ADR(IngombroDestinazioneY_Pos),
						IngombroDestinazioneX_Neg 	:= ADR(IngombroDestinazioneX_Neg),
						IngombroDestinazioneY_Neg 	:= ADR(IngombroDestinazioneY_Neg),
						IngombroDestinazioneZ_Pos 	:= ADR(IngombroDestinazioneZ_Pos),
						IngombroDestinazioneZ_Neg 	:= ADR(IngombroDestinazioneZ_Neg),
						IngombroMaxX_Pos 			:= ADR(IngombroMaxX_Pos),
						IngombroMaxY_Pos 			:= ADR(IngombroMaxY_Pos),
						IngombroMaxX_Neg 			:= ADR(IngombroMaxX_Neg),
						IngombroMaxY_Neg 			:= ADR(IngombroMaxY_Neg),
						IngombroMaxZ_Pos 			:= ADR(IngombroMaxZ_Pos),
						IngombroMaxZ_Neg 			:= ADR(IngombroMaxZ_Neg),
						IngombroY_Pos_0  			:= ADR(IngombroY_Pos_0),		 		
						IngombroY_Neg_180 			:= ADR(IngombroY_Neg_180),
						IngombroY_Neg_0 			:= ADR(IngombroY_Neg_0),	
						IngombroY_Pos_180 			:= ADR(IngombroY_Pos_180),
						ScostamentoVerticalePuntoCentrale := ADR(ScostamentoVerticalePuntoCentrale));





(* Assegnazione quote alla Missione *)
TFWAM_CreaMissione_PrelLastraDaWA(NPosInLavoro				:= Mission^.PPick, //Numero Postazione di lavoro
									Angolo_Destinazione 	:= LatoPrelievo, //Angolo di deposito dell'elemento
									PosizioneAttuale_X      := ModuleAX_X^.Ax^.Status.ActPosition, //Posizione attuale asse X
									TipologiaTraiettoria    := TRAIETTORIA_CON_APPROCCIO,//Forming^[WorkAreaState^[cwa].F].PElement[WorkAreaState^[cwa].P].Trajectory,
									Apprendimento			:= WorkAreaState^[Mission^.PPick].Apprendimento,
									CicloDiPrelievo         := TRUE,
									HmaxElemento			:= WorkAreaState^[Mission^.PPick].Supporto.HMAX,
									Offset_Apprendimento_X 	:= 0,//OffsetApprendimento.Lastra.X, //Offset X Postazione,
									Offset_Apprendimento_Y 	:= OffsetApprendimento.Lastra.Y, //Offset Y Postazione
									Offset_Apprendimento_Z 	:= OffsetApprendimento.Lastra.Z, //Offset Z Postazione
									Offset_Apprendimento_J 	:= 0,//OffsetApprendimento.Lastra.J, //Offset J Postazione

									Quota_PostX				:= WorkArea^[Mission^.PPick].X, //Quota X Postazione
									Quota_PostY				:= WorkArea^[Mission^.PPick].Y, //Quota Y Postazione
									Quota_PostZ				:= WorkArea^[Mission^.PPick].Z, //Quota Z Postazione
									Quota_PostJ				:= WorkArea^[Mission^.PPick].Rx, //Quota J Postazione
									
									Offset_Postazione_X 	:= WorkAreaOffset^[Mission^.PPick].X, //Offset X Postazione
									Offset_Postazione_Y 	:= WorkAreaOffset^[Mission^.PPick].Y, //Offset Y Postazione
									Offset_Postazione_Z 	:= WorkAreaOffset^[Mission^.PPick].Z, //Offset Z Postazione
									Offset_Postazione_J 	:= WorkAreaOffset^[Mission^.PPick].Rx, //Offset J Postazione
									
									Pallet_DimX				:= WorkAreaState^[Mission^.PPick].Supporto.XDim, //Dimensione X Pallet
									Pallet_DimY				:= WorkAreaState^[Mission^.PPick].Supporto.YDim, //Dimensione Y Pallet
									Pallet_DimZ				:= WorkAreaState^[Mission^.PPick].Supporto.ZDim, //Dimensione Z Pallet
									Pallet_DimBaseUtile		:= WorkAreaState^[Mission^.PPick].Supporto.DimBaseUtile, //Dimensione Z Pallet
									
									Offset_Pallet_X_0		:= 0,//Forming^[WorkAreaState^[Mission^.PPlace].F].Pallet.OFSDE_X0, //Offset X Pallet o Casse
									Offset_Pallet_Y_0		:= 0,//Forming^[WorkAreaState^[Mission^.PPlace].F].Pallet.OFSDE_Y0, //Offset Y Pallet o Casse 
									Offset_Pallet_Z_0		:= OffSetZRecogidaEnAngulo0,//Forming^[WorkAreaState^[Mission^.PPlace].F].Pallet.OFSDE_Z0, //Offset Z Pallet o Casse + è grande + il deposito si distanzia dal supporto
									Offset_Pallet_J_0		:= 0,//Forming^[WorkAreaState^[Mission^.PPlace].F].Pallet.OFSDE_J0, //Offset J Pallet o Casse + è grande + la lastra sarà inclinata verso l'angolo crescente
															   
									Offset_Pallet_X_90		:= 0,//Forming^[WorkAreaState^[Mission^.PPlace].F].Pallet.OFSDE_X90, //Offset X Pallet lato 0-90 
									Offset_Pallet_Y_90		:= 0,//Forming^[WorkAreaState^[Mission^.PPlace].F].Pallet.OFSDE_Y90, //Offset Y Pallet lato 0-90 + è grande + il deposito si distanzia dal supporto
									Offset_Pallet_Z_90		:= 0,//Forming^[WorkAreaState^[Mission^.PPlace].F].Pallet.OFSDE_Z90, //Offset Z Pallet lato 0-90 + è grande + il deposito si distanzia dal supporto
									Offset_Pallet_J_90		:= 0,//Forming^[WorkAreaState^[Mission^.PPlace].F].Pallet.OFSDE_J90, //Offset J Pallet lato 0-90 + è grande + la lastra sarà inclinata in fase di deposito
															  
									Offset_Pallet_X_180		:= 0,//Forming^[WorkAreaState^[Mission^.PPlace].F].Pallet.OFSDE_X180, //Offset X Pallet lato 90-180
									Offset_Pallet_Y_180		:= 0,//Forming^[WorkAreaState^[Mission^.PPlace].F].Pallet.OFSDE_Y180, //Offset Y Pallet lato 90-180 + è grande + il deposito si distanzia dal supporto
									Offset_Pallet_Z_180		:= OffSetZRecogidaEnAngulo180,//Forming^[WorkAreaState^[Mission^.PPlace].F].Pallet.OFSDE_Z180, //Offset Z Pallet lato 90-180 + è grande + il deposito si distanzia dal supporto
									Offset_Pallet_J_180		:= 0,//Forming^[WorkAreaState^[Mission^.PPlace].F].Pallet.OFSDE_J180, //Offset J Pallet lato 90-180 + è grande + la lastra sarà inclinata in fase di deposito
									
									Quota_FormaturaX 		:= 0,//Quota  X da Formatura
									Quota_FormaturaY 		:= ABS(QuotaLastraYRealTimePrelievo),//Quota  Y da Formatura
									Quota_FormaturaZ 		:= QuotaLastraZRealTimePrelievo,//Quota  Z da Formatura
									Quota_FormaturaJ 		:= LatoPrelievo,//Quota  Z da Formatura
									
									Distanza_ApproccioFormaturaX 		:= PickPlaceParameters^.XPickApproach,
									Distanza_ApproccioFormaturaY 		:= PickPlaceParameters^.YPickApproach, 
									Distanza_ApproccioFormaturaZ 		:= PickPlaceParameters^.ZPickApproach,
									Distanza_ApproccioFormaturaJ 		:= PickPlaceParameters^.JPickApproach,
									
									Quota_DestX 			=> Mission^.XPick, //Quota DESTINAZIONE X
									Quota_DestY 			=> Mission^.YPick, //Quota DESTINAZIONE Y
									Quota_DestZ 			=> Mission^.ZPick, //Quota DESTINAZIONE Z
									Quota_DestJ 			=> Mission^.JPick, //Quota DESTINAZIONE J	
									
									Quota_ApproccioDestX 	=> Mission^.XPickApproach, //Quota APPROCCIO di DESTINAZIONE X
									Quota_ApproccioDestY 	=> Mission^.YPickApproach, //Quota APPROCCIO di DESTINAZIONE Y
									Quota_ApproccioDestZ 	=> Mission^.ZPickApproach, //Quota APPROCCIO di DESTINAZIONE Z
									Quota_ApproccioDestJ 	=> Mission^.JPickApproach);//Quota APPROCCIO di DESTINAZIONE J	

//Valorizziamo il preleivo di z a una quota positiva per evitare errori di interferenza									
IF LatoPrelievo = 90 THEN
	IF Mission^.ZPick <= 0 THEN
		Mission^.ZPick := ModuleAX_Z^.AxisPar^.MinPosition;
	END_IF
END_IF 		
//
IF LatoPrelievo = 180 THEN
	
	IF HMI_OffsetDepositoLastra.J180 = 0 OR  HMI_OffsetDepositoLastra.J180 < 0 THEN 
		Mission^.JPick := 180 - 2;
	ELSIF HMI_OffsetDepositoLastra.J180 <= 5 AND   HMI_OffsetDepositoLastra.J180 > 0 THEN 
		Mission^.JPick := 180 - HMI_OffsetDepositoLastra.J180;
	ELSE 
		Mission^.JPick := 180 - 2;	
	END_IF
	


	
	
	
	//IF WorkAreaState^[Mission^.PPick].Apprendimento.Y.Lato180.Stato = APPRENDIMENTO_ESEGUITO THEN
	//	Mission^.YPickApproach	:= MIN(Mission^.YPickApproach,WorkAreaState^[Mission^.PPick].Supporto.YDim + IngombroDestinazioneY_Neg);
	//ELSE
	//	Mission^.YPickApproach	:= WorkArea^[Mission^.PPick].Y + WorkAreaState^[Mission^.PPick].Supporto.YDim + IngombroDestinazioneY_Neg - 50;
	//end_if
	//&&&&&&&&&&&&&&&&&&&&&&&&&&&&&&&&&&&&&&&&&&&&&&&&&&&&&&&&&&&&&&&&&&&&&&&&&&&&&
	//Mission^.YPick 				:= Mission^.YPick - 80 ;	// modificado = 200
	//&&&&&&&&&&&&&&&&&&&&&&&&&&&&&&&&&&&&&&&&&&&&&&&&&&&&&&&&&&&&&&&&&&&&&&&&&&&&&&&&&&&&
	IF WorkareaState^[Mission^.PPick].Supporto.Tipologia = e_Tipo_Pallet.BUNDLE THEN //SE PRELIEVO SU BUNDLE O CASSA
		Y_PuntoPrelievo180 := Mission^.YPick ;
			Z_PuntoPrelievo180Bundle    := Mission^.ZPick ;
		 IF Mission^.YDim  < 1300 THEN
			Mission^.YPick 				:= Mission^.YPick - (80  ) ; //(Dimensioni_Pinza.DimTraveVerticale /2) (*-80*);	// modificado = 200
			Mission^.ZPick				:= Mission^.ZPick + (15 +25) ;
			Mission^.ZPickApproach		:= Mission^.ZPick;
			ELSE
				
			Mission^.YPick 				:= Mission^.YPick (* - (45)*) ; //(Dimensioni_Pinza.DimTraveVerticale /2) (*-80*);	// modificado = 200
 			Mission^.ZPick				:= Mission^.ZPick + 15 ;
			Mission^.ZPickApproach		:= Mission^.ZPick;
		 END_IF
		
	
		
	ELSIF WorkareaState^[Mission^.PPick].Supporto.Tipologia = e_Tipo_Pallet.CAVALLETTO THEN //Se ho in prelievo il supporto di tipo cavalletto	
		Y_PuntoPrelievo180 := Mission^.YPick ;
		Z_PuntoPrelievo180Bundle    := Mission^.ZPick ;
		IF Mission^.YDim  < 1300 THEN
				Mission^.YPick 				:= Mission^.YPick - 10 ; //(Dimensioni_Pinza.DimTraveVerticale -35) ;//(Dimensioni_Pinza.DimTraveVerticale /2) (*-70*)  ;	// modificado = 200
				Mission^.ZPick				:= Mission^.ZPick + (0) ;
				Mission^.ZPickApproach		:= Mission^.ZPick;		
			ELSE
				Mission^.YPick 				:= Mission^.YPick -10(* - 60 *); //(Dimensioni_Pinza.DimTraveVerticale /2) (*-70*)  ;	// modificado = 200
				Mission^.ZPick				:= Mission^.ZPick + 20 ;
				Mission^.ZPickApproach		:= Mission^.ZPick;		
			
		END_IF
		
		
	END_IF

ELSIF LatoPrelievo = 0 THEN
	//Mission^.JPick := 3;
	IF HMI_OffsetDepositoLastra.J0 > 5 THEN 
		Mission^.JPick := 4;
	ELSIF HMI_OffsetDepositoLastra.J0 <> 0 THEN 
		Mission^.JPick := HMI_OffsetDepositoLastra.J0;	
	ELSIF HMI_OffsetDepositoLastra.J0 = 0 THEN 
		Mission^.JPick := 3;	
	END_IF
	Y_PuntoPrelievo0 := Mission^.YPick ;
	
	Z_PuntoPrelievo180Bundle    := Mission^.ZPick ;
	IF Mission^.YDim  < 1300 THEN
			Mission^.YPick 				:= Mission^.YPick -0 ; // + 50 (*+ 50 *);
			Mission^.ZPick				:= Mission^.ZPick + (20) ; // pieza pequeña
			Mission^.ZPickApproach		:= Mission^.ZPick;
		ELSE
			Mission^.YPick 				:= Mission^.YPick  + 100; // + 50 (*+ 50 *);
			Mission^.ZPick				:= Mission^.ZPick + 12 ;
			Mission^.ZPickApproach		:= Mission^.ZPick;	
	END_IF
	
	
	
END_IF											 			
//									
IF TFWAM_CreaMissione_PrelLastraDaWA.Errore.Code > 0 THEN
	Errore := TFWAM_CreaMissione_PrelLastraDaWA.Errore;
	WorkAreaManager^.State 	:= WAMANAGER_NOP;	// setto lo stato del WAMANAGER
	RETURN;//EXIT;
END_IF	

(* Valorizzazione del lato di prelievo nel caso di depostio su cavallina *)
IF WorkareaState^[Mission^.PPlace].Supporto.Tipologia = e_Tipo_Pallet.CAVALLETTO THEN //Se ho in prelievo il supporto di tipo cavalletto
	
	AguloDeDeposito := FunLadoTrabajoCaballete(Piezas_LadoA := 
						HMI_NumeroPezziPresentiCavallete[Mission^.PPlace].HMI_NumeroPezziPresentiPostazione_A_Cavaleto , 
								Piezas_Ladob := HMI_NumeroPezziPresentiCavallete[Mission^.PPlace].HMI_NumeroPezziPresentiPostazione_B_Cavaleto ,
									Recoger := FALSE ,dejar := TRUE, GestionLadoTrabajo := WorkareaState^[Mission^.PPlace].Supporto.TipoTrabajoLado_Cavallete ,
										GestionDescargaCaballete := ADR(GestionCargaCaballete) );
	LatoDeposito := AguloDeDeposito ;

	IF FALSE THEN
		IF FormaturaAFRAMERT[WorkAreaState^[Mission^.PPlace].F].PElement[WorkAreaState^[Mission^.PPlace].P].J > 90 THEN
			LatoDeposito := 180;
		
		ELSIF FormaturaAFRAMERT[WorkAreaState^[Mission^.PPlace].F].PElement[WorkAreaState^[Mission^.PPlace].P].J  < 90 THEN
			LatoDeposito := 0;
		END_IF
	END_IF
	
	
ELSIF WorkareaState^[Mission^.PPlace].Supporto.Tipologia = e_Tipo_Pallet.BUNDLE THEN
	LatoDeposito := 180;
ELSIF WorkareaState^[Mission^.PPlace].Supporto.Tipologia <> e_Tipo_Pallet.CAVALLETTO AND WorkareaState^[Mission^.PPlace].Supporto.Tipologia <> e_Tipo_Pallet.BUNDLE THEN //Se NON ho in prelievo il supporto di tipo cavalletto
	IF PplaceOld <> Mission^.PPlace THEN 	//Ad ogni cambio di postazione setto il valore del lato iniziale a 0
		TFClearApprendimento(ADR(WorkAreaState^[Mission^.PPlace].Apprendimento));//Pulisco la struttura dell'apprendimento
	END_IF
	LatoDeposito := 90; //Setto il lato di prelievo = 90
	TFWAM_CreaMissione_PrelLastraDaWA.Quota_FormaturaJ := 90;//Assegno la quota di 90° per il prelievo, in questo modo la pinza preleverà in orizzontale
	IF WorkAreaState^[Mission^.PPlace].Apprendimento.Z.Lato90.Stato <> APPRENDIMENTO_ESEGUITO THEN
		WorkAreaState^[Mission^.PPlace].Apprendimento.Z.Lato90.Stato := APPRENDIMENTO_DA_ESEGUIRE;
		IF WorkareaState^[Mission^.PPlace].Supporto.Tipologia = e_Tipo_Pallet.CASSA_STANDARD THEN 
			WorkAreaState^[Mission^.PPlace].Apprendimento.Z.Lato90.QuotaStart 	:= 700;
		ELSE
			WorkAreaState^[Mission^.PPlace].Apprendimento.Z.Lato90.QuotaStart 	:= 700;
		END_IF
	END_IF
END_IF

//Disabilito apprendimento in deposito se disabilitato
IF NOT HMI_AbilitaDepositoPaccoOrrizzontaleConTasteggio AND FALSE THEN
	WorkAreaState^[Mission^.PPlace].Apprendimento.Z.Lato90.Stato := APPRENDIMENTO_DISABILITATO;	
END_IF

//mettiamo un offset sul deposito bundle
IF LatoDeposito = 180 THEN
	TFWAM_CreaMissione_DepLastraDaWA.Offset_Pallet_Y_0 := 0;// HMI_OffsetDepositoLastra.Y0;
	TFWAM_CreaMissione_DepLastraDaWA.Offset_Pallet_Z_0 := 0;//HMI_OffsetDepositoLastra.Z0;
	TFWAM_CreaMissione_DepLastraDaWA.Offset_Pallet_Y_0 := 0;

	TFWAM_CreaMissione_DepLastraDaWA.Offset_Pallet_Y_180 := HMI_OffsetDepositoLastra.Y180;
	TFWAM_CreaMissione_DepLastraDaWA.Offset_Pallet_Z_180 := HMI_OffsetDepositoLastra.Z180;
	TFWAM_CreaMissione_DepLastraDaWA.Offset_Pallet_Z_90  := 0;
	AngoloDepositoLastra := 180; // := 180-1; Modificado 16-6-2025
ELSIF LatoDeposito = 90 THEN
	TFWAM_CreaMissione_DepLastraDaWA.Offset_Pallet_Y_180 := 0;
	TFWAM_CreaMissione_DepLastraDaWA.Offset_Pallet_Z_180 := 0;
	TFWAM_CreaMissione_DepLastraDaWA.Offset_Pallet_Y_180 := 0;
	IF NOT HMI_AbilitaDepositoPaccoOrrizzontaleConTasteggio THEN
		TFWAM_CreaMissione_DepLastraDaWA.Offset_Pallet_Z_90  := (* 30 +*) HMI_OffsetDepositoLastra.Z90; // quitado el ´30
	ELSE
		TFWAM_CreaMissione_DepLastraDaWA.Offset_Pallet_Z_90  := 0;
	END_IF
	AngoloDepositoLastra := 90;
ELSIF LatoDeposito = 0 THEN
	TFWAM_CreaMissione_DepLastraDaWA.Offset_Pallet_Y_180 := 0;
	TFWAM_CreaMissione_DepLastraDaWA.Offset_Pallet_Z_180 := 0;
	TFWAM_CreaMissione_DepLastraDaWA.Offset_Pallet_Y_180 := 0;

	//POMGO EL MISMO OFFSET EN Z PARA CAVALINA TANTO EN 0 COMO 180 
	//@@@@@@@@@@@@@@@@@@@@@@Para Quitar@@@@@@@@@@@@@@@@@@@@@@@@@@@@@@@@@@@@@@@@@@@@@@@
	//HMI_OffsetDepositoLastra.Z0 :=HMI_OffsetDepositoLastra.Z180 +10 ;
	//@@@@@@@@@@@@@@@@@@@@@@@@@@@@@@@@@@@@@@@@@@@@@@@@@@@@@@@@@@@@@@@@@@@@@
	TFWAM_CreaMissione_DepLastraDaWA.Offset_Pallet_Y_0 := HMI_OffsetDepositoLastra.Y0;
	TFWAM_CreaMissione_DepLastraDaWA.Offset_Pallet_Z_0 := HMI_OffsetDepositoLastra.Z0;
	TFWAM_CreaMissione_DepLastraDaWA.Offset_Pallet_Z_90  := 0;
	AngoloDepositoLastra := 1;
END_IF
// Calculo Del Ingombro Pinza Mision deposito lastra
TFCalcoliIngombroPinza(Mission := Mission,
						WorkAreaManager := WorkAreaManager,
						WorkAreaState := ADR(WorkAreaState),
						ModuleAX_J := ModuleAX_J,
						AngoloRotazioneDestinazionePinza:= AngoloDepositoLastra,//Forming^[WorkAreaState^[Mission^.PPlace].F].PElement[WorkAreaState^[Mission^.PPlace].P].J+2,
						IngombroX_Pos 				:= ADR(IngombroX_Pos),
						IngombroY_Pos 				:= ADR(IngombroY_Pos),
						IngombroX_Neg 				:= ADR(IngombroX_Neg),
						IngombroY_Neg 				:= ADR(IngombroY_Neg),
						IngombroZ_Pos 				:= ADR(IngombroZ_Pos),
						IngombroZ_Neg 				:= ADR(IngombroZ_Neg),
						IngombroY_Tot 				:= ADR(IngombroY_Tot),
						IngombroDestinazioneX_Pos 	:= ADR(IngombroDestinazioneX_Pos),
						IngombroDestinazioneY_Pos 	:= ADR(IngombroDestinazioneY_Pos),
						IngombroDestinazioneX_Neg 	:= ADR(IngombroDestinazioneX_Neg),
						IngombroDestinazioneY_Neg 	:= ADR(IngombroDestinazioneY_Neg),
						IngombroDestinazioneZ_Pos 	:= ADR(IngombroDestinazioneZ_Pos),
						IngombroDestinazioneZ_Neg 	:= ADR(IngombroDestinazioneZ_Neg),
						IngombroMaxX_Pos 			:= ADR(IngombroMaxX_Pos),
						IngombroMaxY_Pos 			:= ADR(IngombroMaxY_Pos),
						IngombroMaxX_Neg 			:= ADR(IngombroMaxX_Neg),
						IngombroMaxY_Neg 			:= ADR(IngombroMaxY_Neg),
						IngombroMaxZ_Pos 			:= ADR(IngombroMaxZ_Pos),
						IngombroMaxZ_Neg 			:= ADR(IngombroMaxZ_Neg),
						IngombroY_Pos_0  			:= ADR(IngombroY_Pos_0),		 		
						IngombroY_Neg_180 			:= ADR(IngombroY_Neg_180),
						IngombroY_Neg_0 			:= ADR(IngombroY_Neg_0),	
						IngombroY_Pos_180 			:= ADR(IngombroY_Pos_180),
						ScostamentoVerticalePuntoCentrale := ADR(ScostamentoVerticalePuntoCentrale));

ScostamentoVerticalePuntoCentrale := ABS(Dimensioni_Pinza.Spessore * COS(deg_to_rad(-90+AngoloDepositoLastra))-Dimensioni_Pinza.Spessore);		
IF HabilitacionFormacionNueva THEN
	FormaturaBundleRT[WorkAreaProductionList^[Mission^.PPlace].NumeroListaAssociata] := FormaturaWa[Mission^.PPlace];
	FormaturaAFRAMERT[WorkAreaProductionList^[Mission^.PPlace].NumeroListaAssociata] := FormaturaWa[Mission^.PPlace];
	;
END_IF

//Z prelievo a seconda della tipologia 
IF WorkareaState^[Mission^.PPlace].Supporto.Tipologia = e_Tipo_Pallet.BUNDLE THEN //Se ho in DEPOSITO il supporto di tipo BUNDLE
	IF LatoDeposito <> 90 THEN
		QuotaLastraYRealTimeDeposito 		:= FormaturaBundleRT[WorkAreaProductionList^[Mission^.PPlace].NumeroListaAssociata].PElement[WorkAreaState^[Mission^.PPlace].P].Y;
		QuotaLastraZRealTimeDeposito 		:= FormaturaBundleRT[WorkAreaProductionList^[Mission^.PPlace].NumeroListaAssociata].PElement[WorkAreaState^[Mission^.PPlace].P].Z;
	ELSE
		Errore.Code := ErrWA_SupportoInPrelivoNonPrevisto;
	END_IF
ELSIF WorkareaState^[Mission^.PPlace].Supporto.Tipologia = e_Tipo_Pallet.CAVALLETTO THEN //Se ho in DEPOSITO il supporto di tipo CAVALLETTO
	IF LatoDeposito = 0 THEN 
		QuotaLastraYRealTimeDeposito 			:= FormaturaAFRAMERT[WorkAreaProductionList^[Mission^.PPlace].NumeroListaAssociata].PElement[WorkAreaState^[Mission^.PPlace].P_Cava.HMI_NumeroPezziPresentiPostazione_A_Cavaleto].CooCavallete.LadoA.CoordenadaFinale_Y;
		QuotaLastraZRealTimeDeposito			:= FormaturaAFRAMERT[WorkAreaProductionList^[Mission^.PPlace].NumeroListaAssociata].PElement[WorkAreaState^[Mission^.PPlace].P_Cava.HMI_NumeroPezziPresentiPostazione_A_Cavaleto].CooCavallete.LadoA.CoordenadaFinale_Z;
	ELSIF LatoDeposito = 180   THEN 
		QuotaLastraYRealTimeDeposito 			:= FormaturaAFRAMERT[WorkAreaProductionList^[Mission^.PPlace].NumeroListaAssociata].PElement[WorkAreaState^[Mission^.PPlace].P_Cava.HMI_NumeroPezziPresentiPostazione_B_Cavaleto].CooCavallete.LadoB.CoordenadaFinale_Y;
		QuotaLastraZRealTimeDeposito			:= FormaturaAFRAMERT[WorkAreaProductionList^[Mission^.PPlace].NumeroListaAssociata].PElement[WorkAreaState^[Mission^.PPlace].P_Cava.HMI_NumeroPezziPresentiPostazione_B_Cavaleto].CooCavallete.LadoB.CoordenadaFinale_Z;
	ELSE
		Errore.Code := ErrWA_SupportoInPrelivoNonPrevisto;	
	END_IF

	IF FALSE THEN 
		IF LatoDeposito <> 90 THEN
			QuotaLastraYRealTimeDeposito 		:= FormaturaAFRAMERT[WorkAreaProductionList^[Mission^.PPlace].NumeroListaAssociata].PElement[WorkAreaState^[Mission^.PPlace].P].Y;
			QuotaLastraZRealTimeDeposito 		:= FormaturaAFRAMERT[WorkAreaProductionList^[Mission^.PPlace].NumeroListaAssociata].PElement[WorkAreaState^[Mission^.PPlace].P].Z;
		ELSE
			Errore.Code := ErrWA_SupportoInPrelivoNonPrevisto;
		END_IF
	END_IF
	
	
	
ELSE
	QuotaLastraZRealTimeDeposito := Forming^[WorkAreaState^[Mission^.PPlace].F].PElement[WorkAreaState^[Mission^.PPlace].P].Z;
	QuotaLastraYRealTimeDeposito := ABS(Forming^[WorkAreaState^[Mission^.PPlace].F].PElement[WorkAreaState^[Mission^.PPlace].P].Y);
END_IF	

IF WorkAreaState^[Mission^.PPlace].Supporto.Tipologia = CAVALLETTO THEN
	OffSetY180Cavallete := 0 ;	
	ELSE 
	OffSetY180Cavallete := 0 ;	
	
END_IF


(* Valorizzazione quote di deposito Ciclo Lastra *)
TFWAM_CreaMissione_DepLastraDaWA(NPosInLavoro			:= Mission^.PPlace, //Numero Postazione di lavoro
								Angolo_Destinazione 	:= LatoDeposito, //Angolo di deposito dell'elemento
								PosizioneAttuale_X      := ModuleAX_X^.Ax^.Status.ActPosition, //Posizione attuale asse X
								TipologiaTraiettoria    := TRAIETTORIA_CON_APPROCCIO,//Forming^[WorkAreaState^[cwa].F].PElement[WorkAreaState^[cwa].P].Trajectory,
								Apprendimento			:= WorkAreaState^[Mission^.PPlace].Apprendimento,
								CicloDiPrelievo         := FALSE,
								HmaxElemento			:= WorkAreaState^[Mission^.PPlace].Supporto.HMAX,
								
								Offset_Apprendimento_X 	:= 0,//OffsetApprendimento.Lastra.X, //Offset X Postazione,
								Offset_Apprendimento_Y 	:= TO_REAL(OffsetApprendimento.Lastra.Y), //Offset Y Postazione
								Offset_Apprendimento_Z 	:= TO_REAL(Forming^[WorkAreaState^[Mission^.PPlace].F].PElement[WorkAreaState^[Mission^.PPlace].P].ZDim + OffsetApprendimento.Lastra.Z), //Offset Z Postazione
								Offset_Apprendimento_J 	:= 0,//OffsetApprendimento.Lastra.J, //Offset J Postazione

								Quota_PostX				:= WorkArea^[Mission^.PPlace].X, //Quota X Postazione
								Quota_PostY				:= WorkArea^[Mission^.PPlace].Y, //Quota Y Postazione
								Quota_PostZ				:= WorkArea^[Mission^.PPlace].Z, //Quota Z Postazione
								Quota_PostJ				:= WorkArea^[Mission^.PPlace].Rx, //Quota J Postazione
								
								Offset_Postazione_X 	:= WorkAreaOffset^[Mission^.PPlace].X, //Offset X Postazione
								Offset_Postazione_Y 	:= WorkAreaOffset^[Mission^.PPlace].Y, //Offset Y Postazione
								Offset_Postazione_Z 	:= WorkAreaOffset^[Mission^.PPlace].Z, //Offset Z Postazione
								Offset_Postazione_J 	:= WorkAreaOffset^[Mission^.PPlace].Rx, //Offset J Postazione
								
								Pallet_DimX				:= WorkAreaState^[Mission^.PPlace].Supporto.XDim, //Dimensione X Pallet
								Pallet_DimY				:= WorkAreaState^[Mission^.PPlace].Supporto.YDim, //Dimensione Y Pallet
								Pallet_DimZ				:= WorkAreaState^[Mission^.PPlace].Supporto.ZDim, //Dimensione Z Pallet
								
								Offset_Pallet_X_0		:= 0,//Forming^[WorkAreaState^[Mission^.PPlace].F].Pallet.OFSDE_X0, //Offset X Pallet o Casse
								//Offset_Pallet_Y_0		:= 0,//Forming^[WorkAreaState^[Mission^.PPlace].F].Pallet.OFSDE_Y0, //Offset Y Pallet o Casse 
								//Offset_Pallet_Z_0		:= 0,//Forming^[WorkAreaState^[Mission^.PPlace].F].Pallet.OFSDE_Z0, //Offset Z Pallet o Casse + è grande + il deposito si distanzia dal supporto
								Offset_Pallet_J_0		:= 0,//Forming^[WorkAreaState^[Mission^.PPlace].F].Pallet.OFSDE_J0, //Offset J Pallet o Casse + è grande + la lastra sarà inclinata verso l'angolo crescente
														   
								Offset_Pallet_X_90		:= 0,//Forming^[WorkAreaState^[Mission^.PPlace].F].Pallet.OFSDE_X90, //Offset X Pallet lato 0-90 
								Offset_Pallet_Y_90		:= 0,//Forming^[WorkAreaState^[Mission^.PPlace].F].Pallet.OFSDE_Y90, //Offset Y Pallet lato 0-90 + è grande + il deposito si distanzia dal supporto
								//Offset_Pallet_Z_90		:= 0,//Forming^[WorkAreaState^[Mission^.PPlace].F].Pallet.OFSDE_Z90, //Offset Z Pallet lato 0-90 + è grande + il deposito si distanzia dal supporto
								Offset_Pallet_J_90		:= 0,//Forming^[WorkAreaState^[Mission^.PPlace].F].Pallet.OFSDE_J90, //Offset J Pallet lato 0-90 + è grande + la lastra sarà inclinata in fase di deposito
														  
								Offset_Pallet_X_180		:= 0,//Forming^[WorkAreaState^[Mission^.PPlace].F].Pallet.OFSDE_X180, //Offset X Pallet lato 90-180
								//Offset_Pallet_Y_180		:= OffSetY180Cavallete , //0,//Forming^[WorkAreaState^[Mission^.PPlace].F].Pallet.OFSDE_Y180, //Offset Y Pallet lato 90-180 + è grande + il deposito si distanzia dal supporto
								//Offset_Pallet_Z_180		:= 0,//Forming^[WorkAreaState^[Mission^.PPlace].F].Pallet.OFSDE_Z180, //Offset Z Pallet lato 90-180 + è grande + il deposito si distanzia dal supporto
								Offset_Pallet_J_180		:= 0,//Forming^[WorkAreaState^[Mission^.PPlace].F].Pallet.OFSDE_J180, //Offset J Pallet lato 90-180 + è grande + la lastra sarà inclinata in fase di deposito
								
								Quota_FormaturaX 		:= Forming^[WorkAreaState^[Mission^.PPlace].F].PElement[WorkAreaState^[Mission^.PPlace].P].X, //Quota Deposito X da Formatura
								Quota_FormaturaY 		:= ABS(QuotaLastraYRealTimeDeposito),//ABS(Forming^[WorkAreaState^[Mission^.PPlace].F].PElement[WorkAreaState^[Mission^.PPlace].P].Y), //Quota Deposito Y da Formatura
								Quota_FormaturaZ 		:= ABS(QuotaLastraZRealTimeDeposito),//Forming^[WorkAreaState^[Mission^.PPlace].F].PElement[WorkAreaState^[Mission^.PPlace].P].Z, //Quota Deposito Z da Formatura
								Quota_FormaturaJ 		:= AngoloDepositoLastra,//Forming^[WorkAreaState^[Mission^.PPlace].F].PElement[WorkAreaState^[Mission^.PPlace].P].J, //Quota Deposito Z da Formatura
								
								Distanza_ApproccioFormaturaX 		:= 0,//PickPlaceParameters^.XPlaceApproach,
								Distanza_ApproccioFormaturaY 		:= PickPlaceParameters^.YPlaceApproach, 
								Distanza_ApproccioFormaturaZ 		:= PickPlaceParameters^.ZPlaceApproach,
								Distanza_ApproccioFormaturaJ 		:= 0,//PickPlaceParameters^.JPlaceApproach,

								Quota_DestX 			=> Mission^.XPlace, //Quota DESTINAZIONE X
								Quota_DestY 			=> Mission^.YPlace, //Quota DESTINAZIONE Y
								Quota_DestZ 			=> Mission^.ZPlace, //Quota DESTINAZIONE Z
								Quota_DestJ 			=> Mission^.JPlace, //Quota DESTINAZIONE J	
								
								Quota_ApproccioDestX 	=> Mission^.XPlaceApproach, //Quota APPROCCIO di DESTINAZIONE X
								Quota_ApproccioDestY 	=> Mission^.YPlaceApproach, //Quota APPROCCIO di DESTINAZIONE Y
								Quota_ApproccioDestZ 	=> Mission^.ZPlaceApproach, //Quota APPROCCIO di DESTINAZIONE Z
								Quota_ApproccioDestJ 	=> Mission^.JPlaceApproach);//Quota APPROCCIO di DESTINAZIONE J	

//memorizzo la postazione di deposito
PplaceOld := Mission^.PPlace;
								
IF LatoDeposito = 90 AND WorkAreaState^[Mission^.PPlace].Apprendimento.Z.Lato90.Stato <> APPRENDIMENTO_ESEGUITO THEN
	Mission^.ZPlace := Mission^.ZPlace-50;
END_IF						
															
(* Passo alla pinza i valori di dimensione della lastra *)
ModulePinza^.ElementoInPrelievo.XDim := Mission^.XDim;
ModulePinza^.ElementoInPrelievo.YDim := Mission^.YDim;
ModulePinza^.ElementoInPrelievo.ZDim := Mission^.ZDim;
ModulePinza^.ElementoInPrelievo.Typology := LASTRA;

(* Se il FB di calcolo delle quote Restituisce un errore Mi fermo, altrimenti Eseguo la missione *)
IF TFWAM_CreaMissione_DepLastraDaWA.Errore.Code > 0 THEN
	Errore := TFWAM_CreaMissione_DepLastraDaWA.Errore;
	WorkAreaManager^.State 	:= WAMANAGER_NOP;	// setto lo stato del WAMANAGER
	RestoreCWA^ := TRUE;
	PreviousPWA^ := pwa;
	RETURN;//EXIT;
ELSE
	//IF Mission^.PPick = NumPostazioneDiPareggiatura THEN
	//	WorkAreaManager^.State 	:= WAMANAGER_CICLO_PRELIEVO_LASTRA_DA_PAREGGIATORE_RUN;
	//ELSE
		WorkAreaManager^.State 	:= WAMANAGER_CICLO_PRELIEVO_LASTRA_WA_RUN;
	//END_IF
	RestoreCWA^ := TRUE;
	PreviousPWA^ := pwa;
	RETURN;//EXIT;
END_IF

(* Setto l'uscita che mi determina il deposito del primo pacco in lenta *)
IF WorkAreaState^[Mission^.PPick].Slow = 1 THEN
	DepositoPaccoInLenta := TRUE;
END_IF
END_ACTION

ACTION PREL_DA_PAREGGIATORE_END:
(* Se era settata la velocità lenta di Prelievo pacco, questa viene resettata *)
IF WorkAreaState^[Mission^.PPick].Slow = 1 THEN
	WorkAreaState^[Mission^.PPick].Slow := 0;
	DepositoPaccoInLenta := FALSE;
END_IF
(* Aggiorno la struttura delle Lastre Presenti *)
Mission^.Slab := WorkAreaState^[Mission^.PPick].Slab[NLastraDaPrelevare];
(* Decremento WorkArea^[cwa].P (P=P-1) *)
WorkAreaState^[Mission^.PPick].P := WorkAreaState^[Mission^.PPick].P - 1;

WorkAreaManager^.State 	:= WAMANAGER_CICLO_DEPOSITO_LASTRA_WA_RUN;
RestoreCWA^ := TRUE;
PreviousPWA^ := pwa;
RETURN;//EXIT;
END_ACTION

ACTION PREL_DA_PAREGGIATORE_RUN:
	
IF Mission^.State = MISSION_STATE_PRELIEVO_LASTRA_DA_PAREGGIATORE_RUN THEN
	WorkAreaManager^.State 	:= WAMANAGER_CICLO_PRELIEVO_LASTRA_DA_PAREGGIATORE_RUN;
ELSIF Mission^.State = MISSION_STATE_PRELIEVO_LASTRA_DA_PAREGGIATORE_END THEN
	WorkAreaManager^.State 	:= WAMANAGER_CICLO_PRELIEVO_LASTRA_DA_PAREGGIATORE_END;
ELSIF Mission^.State = MISSION_STATE_ERROR THEN
	;
END_IF
END_ACTION

ACTION PREL_FALDA_END:
CASE TIPO_MAGAZZINO_FALDE OF 
	(* Se il magazzino delle falde è PickPoint *)
	MAGAZZINO_FALDE_IN_PP: 		
		IF WorkPickPoint^[Mission^.PPick].Tipologia = MAGAZZINO_FALDE THEN
			IF WorkPickPoint^[Mission^.PPick].Learned_Z > WorkPickPoint^[Mission^.PPick].Z + Mission^.ZDim THEN
				WorkPickPoint^[Mission^.PPick].Learn_Z 		:= ALTEZZA_CATASTA_FALDE;
				WorkPickPoint^[Mission^.PPick].Learned_Z 	:= ModuleAX_Z^.Ax^.Status.ActPosition; 
				WorkPickPoint^[Mission^.PPick].DoLearn_Z	:= APPRENDIMENTO_ESEGUITO;
			ELSE
				WorkPickPoint^[Mission^.PPick].Learn_Z 		:= ALTEZZA_CATASTA_FALDE;
				WorkPickPoint^[Mission^.PPick].Learned_Z 	:= ALTEZZA_CATASTA_FALDE;
				WorkPickPoint^[Mission^.PPick].DoLearn_Z 	:= APPRENDIMENTO_DA_ESEGUIRE;
				//WorkAreaState^[Mission^.PPick].State := WORKAREA_STATE_OCCUPIED_ENDED;	
			END_IF
		ELSE
			Errore.Code := ErrWAM_PickPoint_NoMagazzinoFalde;//Errore, Il Pick Point, non è di tipo Magazzino Falde
			RETURN;//EXIT;
		END_IF
	(* Se il magazzino delle falde è una WorkArea *)
	MAGAZZINO_FALDE_IN_WA:	
		IF WorkArea^[Mission^.PPick].Typology = TYPOLOGY_LAYER THEN
			IF WorkAreaState^[Mission^.PPick].H > WorkArea^[Mission^.PPick].Z + Mission^.ZDim THEN
				WorkAreaState^[Mission^.PPick].H 			:= ModuleAX_Z^.Ax^.Status.ActPosition; 
				WorkAreaState^[Mission^.PPick].Apprendimento.Z.Lato0.QuotaStart 	:= ALTEZZA_CATASTA_FALDE;
				WorkAreaState^[Mission^.PPick].Apprendimento.Z.Lato0.QuotaRilevata 	:= ModuleAX_Z^.Ax^.Status.ActPosition;
				WorkAreaState^[Mission^.PPick].Apprendimento.Z.Lato0.Stato		 	:= APPRENDIMENTO_ESEGUITO;
			ELSE
				WorkAreaState^[Mission^.PPick].H 			:= WorkArea^[Mission^.PPick].Z;
				WorkAreaState^[Mission^.PPick].Apprendimento.Z.Lato0.QuotaStart 	:= ALTEZZA_CATASTA_FALDE;
				WorkAreaState^[Mission^.PPick].Apprendimento.Z.Lato0.QuotaRilevata 	:= ALTEZZA_CATASTA_FALDE;
				WorkAreaState^[Mission^.PPick].Apprendimento.Z.Lato0.Stato		 	:= APPRENDIMENTO_DA_ESEGUIRE;
				//WorkAreaState^[Mission^.PPick].State := WORKAREA_STATE_OCCUPIED_ENDED;	
			END_IF
			(* Aggiorno la struttura delle Lastre Presenti *)
			Mission^.Slab := WorkAreaState^[Mission^.PPick].Slab[NLastraDaPrelevare];
			(* Decremento WorkArea^[cwa].P (P=P-1) *)
			WorkAreaState^[Mission^.PPick].P := WorkAreaState^[Mission^.PPick].P - 1;
		ELSE
			Errore.Code := ErrWAM_WorkArea_NoMagazzinoFalde; // Errore, la WorkArea non è di tipo Magazzino Falde
			RETURN;//	EXIT;
		END_IF
ELSE
	Errore.Code := ErrWAM_TipologiaMagazzinoFaldaNONRiconosciuta;// Errore, Nell'impianto è stata impostata una tipologia di magazzino falde non prevista!!!
	RETURN;//EXIT;		
END_CASE
WorkAreaManager^.State 	:= WAMANAGER_CICLO_DEPOSITO_FALDA_RUN;
RestoreCWA^ := TRUE;
PreviousPWA^ := pwa;
RETURN;//EXIT;
END_ACTION

ACTION PREL_FALDA_RUN:
IF Mission^.State = MISSION_STATE_PRELIEVO_FALDA_RUN THEN
	WorkAreaManager^.State := WAMANAGER_CICLO_PRELIEVO_FALDA_RUN;
ELSIF Mission^.State = MISSION_STATE_PRELIEVO_FALDA_END THEN
	WorkAreaManager^.State := WAMANAGER_CICLO_PRELIEVO_FALDA_END;
	RestoreCWA^ := TRUE;
	PreviousPWA^ := pwa;
	RETURN;//EXIT;
ELSIF Mission^.State = MISSION_STATE_ERROR THEN
	;
END_IF
END_ACTION

ACTION PREL_LASTRA_PP_END:
(* Se era settata la velocità lenta di Prelievo pacco, questa viene resettata *)
IF WorkAreaState^[Mission^.PPick].Slow = 1 THEN
	WorkAreaState^[Mission^.PPick].Slow := 0;
	DepositoPaccoInLenta := FALSE;
END_IF

(* Aggiorno Altezza Pallet su Ultima Lastra depositata *)
(*!!!!!!!!!!! ATTUALMENTE CI BASIAMO SULLE QUOTE INVIATE DA HMI PER IL DEPOSITO E ANDIAMO IN TASTEGGIO, LE CASSE SONO PIU' ALTE DELLA LASTRA DEPOSITATA E 
IN CASO DI CAVALLETTO L'ALTEZZA E' FISSA... QUINDI, NON AGGIORNIAMO NESSUNA ALTEZZA!!!!!*)
(**IF AbilitaAggiornamento_AltezzaWA_ConQuotaAsseZ THEN
	WorkArea^[Mission^.PPlace].H := ModuloAsse_Z.Ax^.Status.ActPosition;
ELSE
	WorkArea^[Mission^.PPlace].H := WorkArea^[Mission^.PPlace].HPL + 
									Forming^[WorkAreaState^[Mission^.PPlace].F].PackXP[WorkAreaState^[Mission^.PPlace].P].Z;
END_IF**)			
CASE TIPOLOGIA_FUNZIONAMENTO_MACCHINA OF
	FUNZIONAMENTO_PALLETTIZZATORE:
									WorkAreaManager^.State 	:= WAMANAGER_CICLO_DEPOSITO_LASTRA_PP_RUN;
									RestoreCWA^ 	:= TRUE;
									PreviousPWA^ 	:= pwa;
									RETURN;//EXIT;
							
ELSE
	CASE WorkAreaProductionList^[cwa].PElementList[WorkAreaState^[Mission^.PPlace].P].Pareggiatura OF
		(* Se la Pareggiatura della Lastra è Disabilitata *)
		PAREGGIATURA_DISABILITATA:
									WorkAreaManager^.State 	:= WAMANAGER_CICLO_DEPOSITO_LASTRA_PP_RUN;
									RestoreCWA^ := TRUE;
									PreviousPWA^ := pwa;
									RETURN;//EXIT;
									
		(* Se la Pareggiatura della Lastra è Abilitata e da Eseguire *)
		PAREGGIATURA_DA_ESEGUIRE:
									Mission^.PPlace := NumPostazioneDiPareggiatura;
									(* Valorizzazione quote di deposito Ciclo Lastra *)
									TFWAM_CreaMissione_DepLastraDaWA(NPosInLavoro			:= Mission^.PPlace, //Numero Postazione di depositio
																		Angolo_Destinazione 		:= Forming^[WorkAreaState^[Mission^.PPlace].F].PElement[WorkAreaState^[Mission^.PPlace].P].J, //Angolo di deposito dell'elemento
																		PosizioneAttuale_X      := ModuleAX_X^.Ax^.Status.ActPosition, //Posizione attuale asse X
																		TipologiaTraiettoria    := Forming^[WorkAreaState^[cwa].F].PElement[WorkAreaState^[cwa].P].Trajectory,
																			
																		Quota_PostX				:= WorkArea^[Mission^.PPlace].X, //Quota X Postazione
																		Quota_PostY				:= WorkArea^[Mission^.PPlace].Y, //Quota Y Postazione
																		Quota_PostZ				:= WorkArea^[Mission^.PPlace].Z, //Quota Z Postazione
																		Quota_PostJ				:= WorkArea^[Mission^.PPlace].Rx, //Quota J Postazione
																		
																		Offset_Postazione_X 	:= WorkAreaOffset^[Mission^.PPlace].X, //Offset X Postazione
																		Offset_Postazione_Y 	:= WorkAreaOffset^[Mission^.PPlace].Y, //Offset Y Postazione
																		Offset_Postazione_Z 	:= WorkAreaOffset^[Mission^.PPlace].Z, //Offset Z Postazione
																		Offset_Postazione_J 	:= WorkAreaOffset^[Mission^.PPlace].Rx, //Offset J Postazione
																		
																		Pallet_DimX				:= Forming^[WorkAreaState^[Mission^.PPlace].F].Pallet.XDim, //Dimensione X Pallet
																		Pallet_DimY				:= Forming^[WorkAreaState^[Mission^.PPlace].F].Pallet.YDim, //Dimensione Y Pallet
																		Pallet_DimZ				:= Forming^[WorkAreaState^[Mission^.PPlace].F].Pallet.ZDim, //Dimensione Z Pallet
																		
																		Offset_Pallet_X_0		:= Forming^[WorkAreaState^[Mission^.PPlace].F].Pallet.OFSDE_X0, //Offset X Pallet o Casse
																		Offset_Pallet_Y_0		:= Forming^[WorkAreaState^[Mission^.PPlace].F].Pallet.OFSDE_Y0, //Offset Y Pallet o Casse 
																		Offset_Pallet_Z_0		:= Forming^[WorkAreaState^[Mission^.PPlace].F].Pallet.OFSDE_Z0, //Offset Z Pallet o Casse + è grande + il deposito si distanzia dal supporto
																		Offset_Pallet_J_0		:= Forming^[WorkAreaState^[Mission^.PPlace].F].Pallet.OFSDE_J0, //Offset J Pallet o Casse + è grande + la lastra sarà inclinata verso l'angolo crescente
																		
																		Offset_Pallet_X_90		:= Forming^[WorkAreaState^[Mission^.PPlace].F].Pallet.OFSDE_X90, //Offset X Pallet lato 0-90 
																		Offset_Pallet_Y_90		:= Forming^[WorkAreaState^[Mission^.PPlace].F].Pallet.OFSDE_Y90, //Offset Y Pallet lato 0-90 + è grande + il deposito si distanzia dal supporto
																		Offset_Pallet_Z_90		:= Forming^[WorkAreaState^[Mission^.PPlace].F].Pallet.OFSDE_Z90, //Offset Z Pallet lato 0-90 + è grande + il deposito si distanzia dal supporto
																		Offset_Pallet_J_90		:= Forming^[WorkAreaState^[Mission^.PPlace].F].Pallet.OFSDE_J90, //Offset J Pallet lato 0-90 + è grande + la lastra sarà inclinata in fase di deposito
																		
																		Offset_Pallet_X_180		:= Forming^[WorkAreaState^[Mission^.PPlace].F].Pallet.OFSDE_X180, //Offset X Pallet lato 90-180
																		Offset_Pallet_Y_180		:= Forming^[WorkAreaState^[Mission^.PPlace].F].Pallet.OFSDE_Y180, //Offset Y Pallet lato 90-180 + è grande + il deposito si distanzia dal supporto
																		Offset_Pallet_Z_180		:= Forming^[WorkAreaState^[Mission^.PPlace].F].Pallet.OFSDE_Z180, //Offset Z Pallet lato 90-180 + è grande + il deposito si distanzia dal supporto
																		Offset_Pallet_J_180		:= Forming^[WorkAreaState^[Mission^.PPlace].F].Pallet.OFSDE_J180, //Offset J Pallet lato 90-180 + è grande + la lastra sarà inclinata in fase di deposito
																		
																		Quota_FormaturaX 		:= Forming^[WorkAreaState^[Mission^.PPlace].F].PElement[WorkAreaState^[Mission^.PPlace].P].X, //Quota Deposito X da Formatura
																		Quota_FormaturaY 		:= Forming^[WorkAreaState^[Mission^.PPlace].F].PElement[WorkAreaState^[Mission^.PPlace].P].Y, //Quota Deposito Y da Formatura
																		Quota_FormaturaZ 		:= Forming^[WorkAreaState^[Mission^.PPlace].F].PElement[WorkAreaState^[Mission^.PPlace].P].Z, //Quota Deposito Z da Formatura
																		Quota_FormaturaJ 		:= Forming^[WorkAreaState^[Mission^.PPlace].F].PElement[WorkAreaState^[Mission^.PPlace].P].J, //Quota Deposito Z da Formatura
																		
																		Distanza_ApproccioFormaturaX 		:= Forming^[WorkAreaState^[Mission^.PPlace].F].PElement[WorkAreaState^[Mission^.PPlace].P].AX, //Quota Deposito X da Formatura
																		Distanza_ApproccioFormaturaY 		:= Forming^[WorkAreaState^[Mission^.PPlace].F].PElement[WorkAreaState^[Mission^.PPlace].P].AY, //Quota Deposito Y da Formatura
																		Distanza_ApproccioFormaturaZ 		:= Forming^[WorkAreaState^[Mission^.PPlace].F].PElement[WorkAreaState^[Mission^.PPlace].P].AZ, //Quota Deposito Z da Formatura
																		Distanza_ApproccioFormaturaJ 		:= Forming^[WorkAreaState^[Mission^.PPlace].F].PElement[WorkAreaState^[Mission^.PPlace].P].AJ, //Quota Deposito Z da Formatura
																		
																		Quota_DestX 			=> Mission^.XPlace, //Quota DESTINAZIONE X
																		Quota_DestY 			=> Mission^.YPlace, //Quota DESTINAZIONE Y
																		Quota_DestZ 			=> Mission^.ZPlace, //Quota DESTINAZIONE Z
																		Quota_DestJ 			=> Mission^.JPlace, //Quota DESTINAZIONE J	
																		
																		Quota_ApproccioDestX 	=> Mission^.XPlaceApproach, //Quota APPROCCIO di DESTINAZIONE X
																		Quota_ApproccioDestY 	=> Mission^.YPlaceApproach, //Quota APPROCCIO di DESTINAZIONE Y
																		Quota_ApproccioDestZ 	=> Mission^.ZPlaceApproach, //Quota APPROCCIO di DESTINAZIONE Z
																		Quota_ApproccioDestJ 	=> Mission^.JPlaceApproach);//Quota APPROCCIO di DESTINAZIONE J		
			IF TFWAM_CreaMissione_DepLastraDaWA.Errore.Code > 0 THEN
				WorkAreaManager^.State 	:= WAMANAGER_NOP;	// setto lo stato del WAMANAGER
				RETURN;//EXIT;
			ELSE
				WorkAreaManager^.State 	:= WAMANAGER_CICLO_DEPOSITO_LASTRA_SU_PAREGGIATORE_RUN;
				RestoreCWA^ := TRUE;
				PreviousPWA^ := pwa;
				RETURN;//EXIT;
			END_IF	
	ELSE
		;
	END_CASE
END_CASE
END_ACTION

ACTION PREL_LASTRA_PP_RUN:

IF Mission^.State = MISSION_STATE_PRELIEVO_LASTRA_PP_RUN THEN
	;
ELSIF Mission^.State = MISSION_STATE_PRELIEVO_LASTRA_PP_END THEN
	WorkAreaManager^.State 	:= WAMANAGER_CICLO_PRELIEVO_LASTRA_PP_END;
ELSIF Mission^.State = MISSION_STATE_ERROR THEN
	;
END_IF
END_ACTION

ACTION PREL_LASTRA_WA_END:

(* Imposto lo stato dell' apprendimento *)
CASE LatoPrelievo OF			
	0:
		IF WorkAreaState^[Mission^.PPICk].Apprendimento.Y.Lato0.Stato <> APPRENDIMENTO_ESEGUITO THEN
			WorkAreaState^[Mission^.PPICk].Apprendimento.Y.Lato0.Stato := APPRENDIMENTO_ESEGUITO;
			WorkAreaState^[Mission^.PPICk].Apprendimento.Y.Lato0.QuotaRilevata := ModuleAX_Y^.QuotaAsseLetturaTasteggio;
		ELSE
			WorkAreaState^[Mission^.PPICk].Apprendimento.Y.Lato0.QuotaRilevata := ModuleAX_Y^.QuotaAsseLetturaTasteggio;
		END_IF
		
	90:
		IF  WorkAreaState^[Mission^.PPICk].Apprendimento.Z.Lato90.Stato <> APPRENDIMENTO_ESEGUITO THEN
			WorkAreaState^[Mission^.PPICk].Apprendimento.Z.Lato90.Stato 				:= APPRENDIMENTO_ESEGUITO;
			WorkAreaState^[Mission^.PPICk].Apprendimento.Z.Lato90.QuotaRilevata 		:= ModuleAX_Z^.QuotaAsseLetturaTasteggio;
			WorkAreaState^[Mission^.PPICk].Supporto.HMAX 	:=  MAX(WorkAreaState^[Mission^.PPick].Supporto.HMAX,ModuleAX_Z^.QuotaAsseLetturaTasteggio);
			WorkAreaState^[Mission^.PPICk].H 				:=  ModuleAX_Z^.QuotaAsseLetturaTasteggio;
			WorkAreaState^[Mission^.PPICk].HPL 				:=  ModuleAX_Z^.QuotaAsseLetturaTasteggio;	 

		ELSE
			WorkAreaState^[Mission^.PPick].Apprendimento.Z.Lato90.Stato 				:= 	APPRENDIMENTO_ESEGUITO;
			WorkAreaState^[Mission^.PPick].Apprendimento.Z.Lato90.QuotaRilevata 		:=  ModuleAX_Z^.QuotaAsseLetturaTasteggio;
			WorkAreaState^[Mission^.PPick].Supporto.HMAX 	:=  MAX(WorkAreaState^[Mission^.PPick].Supporto.HMAX,ModuleAX_Z^.QuotaAsseLetturaTasteggio);
			WorkAreaState^[Mission^.PPick].H 				:=  ModuleAX_Z^.QuotaAsseLetturaTasteggio;
			WorkAreaState^[Mission^.PPick].HPL 				:=  ModuleAX_Z^.QuotaAsseLetturaTasteggio;	 

		END_IF
		
	180:
		IF WorkAreaState^[Mission^.PPick].Apprendimento.Y.Lato180.Stato <> APPRENDIMENTO_ESEGUITO THEN
			WorkAreaState^[Mission^.PPick].Apprendimento.Y.Lato180.Stato := APPRENDIMENTO_ESEGUITO;
			WorkAreaState^[Mission^.PPick].Apprendimento.Y.Lato180.QuotaRilevata := ModuleAX_Y^.QuotaAsseLetturaTasteggio;
		ELSE
			WorkAreaState^[Mission^.PPick].Apprendimento.Y.Lato180.QuotaRilevata := ModuleAX_Y^.QuotaAsseLetturaTasteggio;
		END_IF
END_CASE

(* Se era settata la velocità lenta di Prelievo pacco, questa viene resettata *)
IF WorkAreaState^[Mission^.PPick].Slow = 1 THEN
	WorkAreaState^[Mission^.PPick].Slow := 0;
	DepositoPaccoInLenta := FALSE;
END_IF

(* Aggiorno Altezza Pallet su Ultima Lastra depositata *)
(*!!!!!!!!!!! ATTUALMENTE CI BASIAMO SULLE QUOTE INVIATE DA HMI PER IL DEPOSITO E ANDIAMO IN TASTEGGIO, LE CASSE SONO PIU' ALTE DELLA LASTRA DEPOSITATA E 
IN CASO DI CAVALLETTO L'ALTEZZA E' FISSA... QUINDI, NON AGGIORNIAMO NESSUNA ALTEZZA!!!!!*)
(**IF AbilitaAggiornamento_AltezzaWA_ConQuotaAsseZ THEN
	WorkArea^[Mission^.PPlace].H := ModuloAsse_Z.Ax^.Status.ActPosition;
ELSE
	WorkArea^[Mission^.PPlace].H := WorkArea^[Mission^.PPlace].HPL + 
									Forming^[WorkAreaState^[Mission^.PPlace].F].PackXP[WorkAreaState^[Mission^.PPlace].P].Z;
END_IF**)


WorkAreaState^[Mission^.PPick].P := WorkAreaState^[Mission^.PPick].P - 1;
IF WorkAreaState^[Mission^.PPick].Supporto.Tipologia = CAVALLETTO THEN 
	IF PosicionJOrigen = 0 THEN 
		WorkAreaState^[Mission^.PPick].P_Cava.HMI_NumeroPezziPresentiPostazione_A_Cavaleto := WorkAreaState^[Mission^.PPick].P_Cava.HMI_NumeroPezziPresentiPostazione_A_Cavaleto -1 ;
	ELSIF PosicionJOrigen = 180 THEN 	
		WorkAreaState^[Mission^.PPick].P_Cava.HMI_NumeroPezziPresentiPostazione_B_Cavaleto := WorkAreaState^[Mission^.PPick].P_Cava.HMI_NumeroPezziPresentiPostazione_B_Cavaleto -1 ;
	END_IF
END_IF

WorkAreaManager^.State 	:= WAMANAGER_CICLO_DEPOSITO_LASTRA_WA_RUN;
RestoreCWA^ := TRUE;
PreviousPWA^ := pwa;
RETURN;//EXIT;
END_ACTION

ACTION PREL_LASTRA_WA_RUN:
IF Mission^.State = MISSION_STATE_PRELIEVO_LASTRA_WA_RUN THEN
	;
ELSIF Mission^.State = MISSION_STATE_PRELIEVO_LASTRA_WA_END THEN
	WorkAreaManager^.State 	:= WAMANAGER_CICLO_PRELIEVO_LASTRA_WA_END;
ELSIF Mission^.State = MISSION_STATE_ERROR THEN
	;
END_IF
END_ACTION

END_FUNCTION_BLOCK

// ---- POUs/TFModules/Moduli TF/TFModulePalletizer_Pinza.TcPOU
FUNCTION_BLOCK TFModulePalletizer_Pinza
VAR_INPUT
	Cmd : CommandBuffer;
	Cfg : Config;
	IN : TFMchinePalletizer_PinzaVentose_IN;
		
	IN_Ax : Module_Palletizer_Ax_IN;
	
	AspirazioneDX1 : POINTER TO TF_VacumOVEM;
	AspirazioneSX1 : POINTER TO TF_VacumOVEM;
	AspirazioneDX2 : POINTER TO TF_VacumOVEM;
	AspirazioneSX2 : POINTER TO TF_VacumOVEM;

	CilindroApertura 			: POINTER TO DC_Cylinder;
	CilindroSbloccoRotazione 	: POINTER TO SC_Cylinder;
	CilindroSbloccoBascolante 	: POINTER TO SC_Cylinder;
	AspirazioneFaldaDX 			: POINTER TO SC_Cylinder;
	AspirazioneFaldaSX 			: POINTER TO SC_Cylinder;
	
	ModuleJ : POINTER TO TFModulePalletizer_Ax;

	ManCmd 				: POINTER TO TFMachinePalletizer_PinzaVentoseManCmd;
	ElementoInPrelievo 	: TFMachinePalletizer_PlaceElement;
	DataElement			: TFMachinePalletizer_DataElement; (* Struttura dati che la macchina acquisisce/trasferisce in fase di pallettizzazione/depallettizazione *)
	PrelievoSuCavallina : BOOL;//indica che il prelievo è su cavallina
	AbilitazioneCilindriTastatori : bool;

	Mission 									: POINTER TO TFMachinePalletizer_Mission;
	AbilitazioneSbloccoRotazione 				: BOOL;//Abilitazione sblocco pinza
	AbilitaAperturaAutomaticaPinza 				: BOOL;//Abilitazione apertura automatica pinza
	AbilitaPrioritaPrelPiasterllaPianiSfalsati 	: BOOL;
	AbilitazioneSbloccoBascolante 				: BOOL;//Abilitazione sblocco bascolante pinza	
END_VAR
VAR_OUTPUT
	CmdExe : CommandExe;
	CmdExd : CommandExe;
	CmdNext : Command;
	CmdLog : CommandLog;
	ProgramLog : ProgrammaLog; 
	State : State;
	StateLog : StateLog;
	Error : Error;
	ErrorLog : ErrorLog;
	Warning : Warning;
	WarningLog : WarningLog;
	OUT : TFMachinePalletizer_PinzaVentose_OUT;
	StatoPinza : TFMachinePalletizer_PinzaState;

END_VAR
VAR
	Power : UINT;
	Init : BOOL;
	Timer : REAL;
	Timeout : REAL;
	TimerAspirazione : REAL;
	ParametersArray : ParametersArray;
	MAN_Actuator : UINT;
	MAN_Cmd : UINT;

	DistanzaFTC0 : REAL;
	DistanzaFTC180 : REAL;

	DistanzaFTC0_2 : REAL;
	DistanzaFTC180_2 : REAL;
	
	TimerPresaPiastrella : REAL;		
	DisattivazioneTotaleAspirazioni : bool;
	FiltroFTCFaldaSX : Signal_Filter;
	FiltroFTCFaldaDX : Signal_Filter;
	
	FTC_FaldaSXFiltrata : BOOL;
	FTC_FaldaDXFiltrata : bool;
	
	AspiraSoloFalde : BOOL;//Se TRUE = si attiva solo l'aspirazione delle falde
	TempoRilascioInDeposito : REAL := 500;
END_VAR

IF NOT Init THEN
	TFCommandBufferClear(ADR(Cmd));
	TFCommandClear(ADR(CmdNext));
	TFCommandExeClear(ADR(CmdExe));
	TFStateUpdate(ADR(State),StateNOP);
	TFErrorClear(ADR(Error));
	TFWarningClear(ADR(Warning));
	Init := TRUE;
	CmdExe.Code := 1;
END_IF

(* Generic Timer - Add here all your Timers *)
TFTimerCall(ADR(Timer),Cfg.TimeBase);
TFTimerCall(ADR(Timeout),Cfg.TimeBase);
TFTimerCall(ADR(TimerPresaPiastrella),Cfg.TimeBase);
TFTimerCall(ADR(TimerAspirazione),Cfg.TimeBase);
(* External To Buffered Command *)
TFCommandToNext(ADR(Cmd),ADR(CmdNext),ADR(CmdExe),ADR(Cfg),ADR(Error),ADR(ErrorLog),ADR(State));

(* Buffered To Exe Command *)
TFCommandToExecution(ADR(CmdNext),ADR(CmdExe),ADR(Error),ADR(ErrorLog),ADR(State),ADR(CmdLog));

(* Chiamata FB *)
AspirazioneDX1^();
AspirazioneSX1^();
AspirazioneDX2^();
AspirazioneSX2^();
CilindroApertura^();
CilindroSbloccoRotazione^();
CilindroSbloccoBascolante^();
AspirazioneFaldaDX^();
AspirazioneFaldaSX^();

DistanzaFTC0 	:= Keyence_LRTB2000C(IN.InKeyence0_Byte0,IN.InKeyence0_Byte1);
DistanzaFTC180 	:= Keyence_LRTB2000C(IN.InKeyence180_Byte0,IN.InKeyence180_Byte1);

DistanzaFTC0_2 	:= Keyence_LRTB2000C(IN.InKeyence0_Byte0_2,IN.InKeyence0_Byte1_2);
DistanzaFTC180_2 	:= Keyence_LRTB2000C(IN.InKeyence180_Byte0_2,IN.InKeyence180_Byte1_2);

FiltroFTCFaldaDX(IN_Signal:=IN.FTC_FaldaDX,FilterTime_ON:=300,FilterTime_OFF:=300,Out_Signal_Filtrato=>FTC_FaldaDXFiltrata);
FiltroFTCFaldaSX(IN_Signal:=IN.FTC_FaldaSX,FilterTime_ON:=300,FilterTime_OFF:=300,Out_Signal_Filtrato=>FTC_FaldaSXFiltrata);


(* Exe Command *)
CASE CmdExe.Code OF

	(* ******************************************************************************************************** *)
	(* Nop  *)
	(* ******************************************************************************************************** *)
	CmdNOP:	;			
	(* ******************************************************************************************************** *)
	(* Stop *)
	(* ******************************************************************************************************** *)
	CmdSTOP:
		CASE CmdExe.CmdCase OF
			
			(* Case 0 *)
			0: 	TFStateUpdate(ADR(State),StateSTOP_RUN);
				TFTimerSet(ADR(Timeout),500,TRUE);
				TFCommandCase(ADR(CmdExe),1,CommandCase_INC);

			(* Case 1 - Clear All Commands*)
			1:	
				TFCommandCase(ADR(CmdExe),100,CommandCase_JMP);
			(* Case 100 *)
			100:TFStateUpdate(ADR(State),StateSTOP_END);
				TFCommandExeClear(ADR(CmdExe));

			ELSE
				TFError(ErrNOCMDCASE,ErrNULL,ADR(CmdExe),ADR(State),ADR(Error),ADR(ErrorLog));
		END_CASE;
	
	(* ******************************************************************************************************** *)
	(* Error Reset *)
	(* ******************************************************************************************************** *)
	CmdRESET:
		CASE CmdExe.CmdCase OF

			(* Case 0 *)
			0: 	TFStateUpdate(ADR(State),StateRESET_RUN);
				TFTimerSet(ADR(Timeout),2000+100,TRUE);
				TFTimerSet(ADR(Timer),2000,TRUE);
				TFCommandCase(ADR(CmdExe),1,CommandCase_INC);
			
			(* Case 1 - RESET COMANDI*)
			1: 
				TFClearAllCmdModulePinzaCompleta(AspirazioneDX1,AspirazioneSX1,AspirazioneDX2,AspirazioneSX2,CilindroApertura,CilindroSbloccoRotazione,CilindroSbloccoBascolante,AspirazioneFaldaDX,AspirazioneFaldaSX);
				TFCommandCase(ADR(CmdExe),1,CommandCase_INC);
			
			(* Case 2 - Invio comando di reset *)
			2:
				AspirazioneDX1^.Command^.ErrorReset 				:= TRUE;	
				AspirazioneSX1^.Command^.ErrorReset 				:= TRUE;	
				AspirazioneDX2^.Command^.ErrorReset 			:= TRUE;	
				AspirazioneSX2^.Command^.ErrorReset 			:= TRUE;	
				CilindroApertura^.Command.ErrorReset 			:= TRUE;	
				CilindroSbloccoRotazione^.Command.ErrorReset 	:= TRUE;	
				CilindroSbloccoBascolante^.Command.ErrorReset 	:= TRUE;	
				AspirazioneFaldaDX^.Command.ErrorReset 			:= TRUE;	
				AspirazioneFaldaSX^.Command.ErrorReset 			:= TRUE;	
				TFCommandCase(ADR(CmdExe),1,CommandCase_INC);
			
			(* Case 3 - Invio comando di reset *)
			3:
				IF AspirazioneDX1^.Status.ErrorResetDone AND
					AspirazioneSX1^.Status.ErrorResetDone AND
					AspirazioneDX2^.Status.ErrorResetDone AND
					AspirazioneSX2^.Status.ErrorResetDone AND
					CilindroApertura^.Status.ErrorResetDone AND
					CilindroSbloccoRotazione^.Status.ErrorResetDone AND
					CilindroSbloccoBascolante^.Status.ErrorResetDone AND
					AspirazioneFaldaDX^.Status.ErrorResetDone AND
					AspirazioneFaldaSX^.Status.ErrorResetDone THEN					
					TFClearAllCmdModulePinzaCompleta(AspirazioneDX1,AspirazioneSX1,AspirazioneDX2,AspirazioneSX2,CilindroApertura,CilindroSbloccoRotazione,CilindroSbloccoBascolante,AspirazioneFaldaDX,AspirazioneFaldaSX);
					TFCommandCase(ADR(CmdExe),99,CommandCase_JMP);
				ELSIF TFTimerDone(ADR(Timer)) THEN
					TFClearAllCmdModulePinzaCompleta(AspirazioneDX1,AspirazioneSX1,AspirazioneDX2,AspirazioneSX2,CilindroApertura,CilindroSbloccoRotazione,CilindroSbloccoBascolante,AspirazioneFaldaDX,AspirazioneFaldaSX);
					TFError(ErrTORESET,ErrNULL,ADR(CmdExe),ADR(State),ADR(Error),ADR(ErrorLog));
				END_IF

			(* Case 99 *)
			99:	TFErrorClear(ADR(Error));
				TFWarningClear(ADR(Warning));
				TFCommandCase(ADR(CmdExe),100,CommandCase_JMP);

			(* Case 100 *)
			100:TFStateUpdate(ADR(State),StateRESET_END);
				TFCommandExeClear(ADR(CmdExe));

			ELSE
				TFError(ErrNOCMDCASE,ErrNULL,ADR(CmdExe),ADR(State),ADR(Error),ADR(ErrorLog));
		END_CASE;

		IF TFTimerDone(ADR(Timeout)) THEN
			TFClearAllCmdModulePinzaCompleta(AspirazioneDX1,AspirazioneSX1,AspirazioneDX2,AspirazioneSX2,CilindroApertura,CilindroSbloccoRotazione,CilindroSbloccoBascolante,AspirazioneFaldaDX,AspirazioneFaldaSX);
			TFError(ErrCMDTIMEOUT,ErrNULL,ADR(CmdExe),ADR(State),ADR(Error),ADR(ErrorLog));
		END_IF
	
	(* ******************************************************************************************************** *)
	(* Power *)
	(* ******************************************************************************************************** *)
	CmdPOWER:
		CASE CmdExe.CmdCase OF
			
			(* Case 0 *)
			0: 	TFStateUpdate(ADR(State),StatePOWER_RUN);
				TFTimerSet(ADR(Timeout),500,TRUE);
				TFCommandCase(ADR(CmdExe),100,CommandCase_JMP);

			1: TFCommandCase(ADR(CmdExe),100,CommandCase_JMP);
			(* Case 100 *)
			100:TFStateUpdate(ADR(State),StatePOWER_END);
				TFCommandExeClear(ADR(CmdExe));

			ELSE
				TFError(ErrNOCMDCASE,ErrNULL,ADR(CmdExe),ADR(State),ADR(Error),ADR(ErrorLog));
		END_CASE
	
	(* ******************************************************************************************************** *)
	(* Home *)
	(* ******************************************************************************************************** *)
	CmdHOME:
		CASE CmdExe.CmdCase OF

			(* Case 0 *)
			0: 	TFStateUpdate(ADR(State),StateHOME_RUN);
				TFTimerSet(ADR(Timeout),3000+200,TRUE);
				TFTimerSet(ADR(Timer),3000,TRUE);
				TFCommandCase(ADR(CmdExe),1,CommandCase_INC);

			(* Case 1 - *)
			1: 
				TFCommandCase(ADR(CmdExe),10,CommandCase_JMP);

			(* Case 10 - Set automatico Soglie *)
			10:
				AspirazioneDX1^.Command^.Aspirazione_ON_ScritturaSoglia 	:= TRUE;
				AspirazioneSX1^.Command^.Aspirazione_ON_ScritturaSoglia 	:= TRUE;
				AspirazioneDX2^.Command^.Aspirazione_ON_ScritturaSoglia 	:= TRUE;
				AspirazioneSX2^.Command^.Aspirazione_ON_ScritturaSoglia 	:= TRUE;
				IF AspirazioneDX1^.Status.CommandDone AND AspirazioneSX1^.Status.CommandDone AND
					AspirazioneDX2^.Status.CommandDone AND AspirazioneSX2^.Status.CommandDone THEN
					AspirazioneDX1^.Command^.Aspirazione_ON_ScritturaSoglia		:= FALSE;
					AspirazioneSX1^.Command^.Aspirazione_ON_ScritturaSoglia		:= FALSE;
					AspirazioneDX2^.Command^.Aspirazione_ON_ScritturaSoglia		:= FALSE;
					AspirazioneSX2^.Command^.Aspirazione_ON_ScritturaSoglia		:= FALSE;
					TFCommandCase(ADR(CmdExe),100,CommandCase_JMP);
				ELSIF TFTimerDone(ADR(Timer)) THEN
					AspirazioneDX1^.Command^.Aspirazione_ON_ScritturaSoglia		:= FALSE;
					AspirazioneSX1^.Command^.Aspirazione_ON_ScritturaSoglia		:= FALSE;
					AspirazioneDX2^.Command^.Aspirazione_ON_ScritturaSoglia		:= FALSE;
					AspirazioneSX2^.Command^.Aspirazione_ON_ScritturaSoglia		:= FALSE;
					TFError(ErrTOHOME,ErrNULL,ADR(CmdExe),ADR(State),ADR(Error),ADR(ErrorLog));
				END_IF
			
	
			(* Case 100 *)
			100:TFStateUpdate(ADR(State),StateHOME_END);
				TFCommandExeClear(ADR(CmdExe));

			ELSE
				TFError(ErrNOCMDCASE,ErrNULL,ADR(CmdExe),ADR(State),ADR(Error),ADR(ErrorLog));
		END_CASE;
		
		IF AspirazioneDX1^.Status.ErrorID <> ErrNULL THEN
			TFClearAllCmdModulePinzaCompleta(AspirazioneDX1,AspirazioneSX1,AspirazioneDX2,AspirazioneSX2,CilindroApertura,CilindroSbloccoRotazione,CilindroSbloccoBascolante,AspirazioneFaldaDX,AspirazioneFaldaSX);
			TFError(ErrCYLINDER,AspirazioneDX1^.Status.ErrorID,ADR(CmdExe),ADR(State),ADR(Error),ADR(ErrorLog));
		ELSIF AspirazioneSX1^.Status.ErrorID <> ErrNULL THEN
			TFClearAllCmdModulePinzaCompleta(AspirazioneDX1,AspirazioneSX1,AspirazioneDX2,AspirazioneSX2,CilindroApertura,CilindroSbloccoRotazione,CilindroSbloccoBascolante,AspirazioneFaldaDX,AspirazioneFaldaSX);
			TFError(ErrCYLINDER,AspirazioneSX1^.Status.ErrorID,ADR(CmdExe),ADR(State),ADR(Error),ADR(ErrorLog));
		ELSIF AspirazioneDX2^.Status.ErrorID <> ErrNULL THEN
			TFClearAllCmdModulePinzaCompleta(AspirazioneDX1,AspirazioneSX1,AspirazioneDX2,AspirazioneSX2,CilindroApertura,CilindroSbloccoRotazione,CilindroSbloccoBascolante,AspirazioneFaldaDX,AspirazioneFaldaSX);
			TFError(ErrCYLINDER,AspirazioneDX2^.Status.ErrorID,ADR(CmdExe),ADR(State),ADR(Error),ADR(ErrorLog));
		ELSIF AspirazioneSX2^.Status.ErrorID <> ErrNULL THEN
			TFClearAllCmdModulePinzaCompleta(AspirazioneDX1,AspirazioneSX1,AspirazioneDX2,AspirazioneSX2,CilindroApertura,CilindroSbloccoRotazione,CilindroSbloccoBascolante,AspirazioneFaldaDX,AspirazioneFaldaSX);
			TFError(ErrCYLINDER,AspirazioneSX2^.Status.ErrorID,ADR(CmdExe),ADR(State),ADR(Error),ADR(ErrorLog));
		ELSIF CilindroApertura^.Status.ErrorID <> ErrNULL THEN
			TFClearAllCmdModulePinzaCompleta(AspirazioneDX1,AspirazioneSX1,AspirazioneDX2,AspirazioneSX2,CilindroApertura,CilindroSbloccoRotazione,CilindroSbloccoBascolante,AspirazioneFaldaDX,AspirazioneFaldaSX);
			TFError(ErrCYLINDER,CilindroApertura^.Status.ErrorID,ADR(CmdExe),ADR(State),ADR(Error),ADR(ErrorLog));
		ELSIF CilindroSbloccoRotazione^.Status.ErrorID <> ErrNULL THEN
			TFClearAllCmdModulePinzaCompleta(AspirazioneDX1,AspirazioneSX1,AspirazioneDX2,AspirazioneSX2,CilindroApertura,CilindroSbloccoRotazione,CilindroSbloccoBascolante,AspirazioneFaldaDX,AspirazioneFaldaSX);
			TFError(ErrCYLINDER,CilindroSbloccoRotazione^.Status.ErrorID,ADR(CmdExe),ADR(State),ADR(Error),ADR(ErrorLog));
		ELSIF AspirazioneFaldaDX^.Status.ErrorID <> ErrNULL THEN
			TFClearAllCmdModulePinzaCompleta(AspirazioneDX1,AspirazioneSX1,AspirazioneDX2,AspirazioneSX2,CilindroApertura,CilindroSbloccoRotazione,CilindroSbloccoBascolante,AspirazioneFaldaDX,AspirazioneFaldaSX);
			TFError(ErrCYLINDER,AspirazioneFaldaDX^.Status.ErrorID,ADR(CmdExe),ADR(State),ADR(Error),ADR(ErrorLog));
		ELSIF AspirazioneFaldaSX^.Status.ErrorID <> ErrNULL THEN
			TFClearAllCmdModulePinzaCompleta(AspirazioneDX1,AspirazioneSX1,AspirazioneDX2,AspirazioneSX2,CilindroApertura,CilindroSbloccoRotazione,CilindroSbloccoBascolante,AspirazioneFaldaDX,AspirazioneFaldaSX);
			TFError(ErrCYLINDER,AspirazioneFaldaSX^.Status.ErrorID,ADR(CmdExe),ADR(State),ADR(Error),ADR(ErrorLog));
		ELSIF TFTimerDone(ADR(Timeout)) THEN
			TFClearAllCmdModulePinzaCompleta(AspirazioneDX1,AspirazioneSX1,AspirazioneDX2,AspirazioneSX2,CilindroApertura,CilindroSbloccoRotazione,CilindroSbloccoBascolante,AspirazioneFaldaDX,AspirazioneFaldaSX);
			TFError(ErrCMDTIMEOUT,ErrNULL,ADR(CmdExe),ADR(State),ADR(Error),ADR(ErrorLog));
		END_IF

	(* ******************************************************************************************************** *)
	(* Manual *)
	(* ******************************************************************************************************** *)
	CmdMAN:
		CASE CmdExe.CmdCase OF
			(* Case 0 *)
			0: 	TFStateUpdate(ADR(State),StateMAN_RUN);
				TFTimerSet(ADR(Timeout),3000,TRUE);
				IF TFCommandParRead(CmdExe.Cmd.Parameter,ADR(ParametersArray),2) THEN
					MAN_Actuator	:= STRING_TO_UINT(ParametersArray.Parameters[0]);
					MAN_Cmd		:= STRING_TO_UINT(ParametersArray.Parameters[1]);
				ELSE
					TFError(ErrCMDPARNUM,ErrNULL,ADR(CmdExe),ADR(State),ADR(Error),ADR(ErrorLog));
					RETURN;
				END_IF;

				CASE MAN_Actuator OF
					(* Case 0..99 for Actuators *)
					(* Case 100..199  for Axis *)

					(* Case Nop *)
					0:	;

					(* Case 1: *)
					1:	CASE MAN_Cmd OF
							0:	;
							
							(* Case 10: Apertura Pinza *)
							10:	
								CilindroApertura^.Command.Activation 	:= TRUE;
								CilindroApertura^.Command.Deactivation 	:= FALSE;
								TFTimerSet(ADR(Timeout),30000,TRUE);
								TFCommandCase(ADR(CmdExe),10,CommandCase_JMP);
								
							(* Case 11: Chiusura Pinza *)
							11:	
								CilindroApertura^.Command.Activation 	:= FALSE;
								CilindroApertura^.Command.Deactivation 	:= TRUE;
								TFTimerSet(ADR(Timeout),30000,TRUE);
								TFCommandCase(ADR(CmdExe),10,CommandCase_JMP);

							(* Case 20: Sgancio Sblocco Rotazione *)
							20:	
								CilindroSbloccoRotazione^.Command.Activation 	:= TRUE;
								CilindroSbloccoRotazione^.Command.Deactivation 	:= FALSE;
								TFTimerSet(ADR(Timeout),3000,TRUE);
								TFCommandCase(ADR(CmdExe),20,CommandCase_JMP);
								
							(* Case 21: Aggancio Sblocco Rotazione *)
							21:	
								CilindroSbloccoRotazione^.Command.Activation 	:= FALSE;
								CilindroSbloccoRotazione^.Command.Deactivation 	:= TRUE;
								TFTimerSet(ADR(Timeout),3000,TRUE);
								TFCommandCase(ADR(CmdExe),20,CommandCase_JMP);

							(* Case 30: Ativazione Aspirazione Falda DX *)
							30:	
								AspirazioneFaldaDX^.Command.Activation 		:= TRUE;
								AspirazioneFaldaDX^.Command.Deactivation 	:= FALSE;
								TFTimerSet(ADR(Timeout),3000,TRUE);
								TFCommandCase(ADR(CmdExe),30,CommandCase_JMP);
								
							(* Case 31: Disattivazione Aspirazione Falda DX *)
							31:	
								AspirazioneFaldaDX^.Command.Activation 		:= FALSE;
								AspirazioneFaldaDX^.Command.Deactivation 	:= TRUE;
								TFTimerSet(ADR(Timeout),3000,TRUE);
								TFCommandCase(ADR(CmdExe),30,CommandCase_JMP);
								
							(* Case 40: Ativazione Aspirazione Falda SX *)
							40:	
								AspirazioneFaldaSX^.Command.Activation 		:= TRUE;
								AspirazioneFaldaSX^.Command.Deactivation 	:= FALSE;

								TFTimerSet(ADR(Timeout),3000,TRUE);
								TFCommandCase(ADR(CmdExe),40,CommandCase_JMP);
								
							(* Case 41: Disattivazione Aspirazione Falda SX *)
							41:	
								AspirazioneFaldaSX^.Command.Activation 		:= FALSE;
								AspirazioneFaldaSX^.Command.Deactivation 	:= TRUE;

								TFTimerSet(ADR(Timeout),3000,TRUE);
								TFCommandCase(ADR(CmdExe),40,CommandCase_JMP);

							(* Case 50: Ativazione Aspirazione SX *)
							50:	
								AspirazioneSX1^.Command^.Aspirazione_ON 	:= TRUE;
								AspirazioneSX1^.Command^.Aspirazione_OFF := FALSE;

								AspirazioneDX1^.Command^.Aspirazione_ON 	:= TRUE;
								AspirazioneDX1^.Command^.Aspirazione_OFF := FALSE;

								AspirazioneSX2^.Command^.Aspirazione_ON 	:= TRUE;
								AspirazioneSX2^.Command^.Aspirazione_OFF := FALSE;

								AspirazioneDX2^.Command^.Aspirazione_ON 	:= TRUE;
								AspirazioneDX2^.Command^.Aspirazione_OFF := FALSE;

								TFTimerSet(ADR(Timeout),3000,TRUE);
								TFCommandCase(ADR(CmdExe),50,CommandCase_JMP);
								
							(* Case 51: Disattivazione Aspirazione SX *)
							51:	
								AspirazioneSX1^.Command^.Aspirazione_ON 	:= FALSE;
								AspirazioneSX1^.Command^.Aspirazione_OFF := TRUE;
								AspirazioneSX2^.Command^.Aspirazione_ON 	:= FALSE;
								AspirazioneSX2^.Command^.Aspirazione_OFF := TRUE;
								TFTimerSet(ADR(Timeout),3000,TRUE);
								TFCommandCase(ADR(CmdExe),50,CommandCase_JMP);

							(* Case 60: Ativazione Aspirazione DX *)
							60:	
								AspirazioneDX1^.Command^.Aspirazione_ON 	:= TRUE;
								AspirazioneDX1^.Command^.Aspirazione_OFF := FALSE;
								AspirazioneDX2^.Command^.Aspirazione_ON 	:= TRUE;
								AspirazioneDX2^.Command^.Aspirazione_OFF := FALSE;
								AspirazioneSX1^.Command^.Aspirazione_ON 	:= TRUE;
								AspirazioneSX1^.Command^.Aspirazione_OFF := FALSE;
								AspirazioneSX2^.Command^.Aspirazione_ON 	:= TRUE;
								AspirazioneSX2^.Command^.Aspirazione_OFF := FALSE;
								TFTimerSet(ADR(Timeout),3000,TRUE);
								TFCommandCase(ADR(CmdExe),60,CommandCase_JMP);
								
							(* Case 61: Disattivazione Aspirazione SX *)
							61:	
								AspirazioneDX1^.Command^.Aspirazione_ON 	:= FALSE;
								AspirazioneDX1^.Command^.Aspirazione_OFF := TRUE;
								AspirazioneSX1^.Command^.Aspirazione_ON 	:= FALSE;
								AspirazioneSX1^.Command^.Aspirazione_OFF := TRUE;
								AspirazioneDX2^.Command^.Aspirazione_ON 	:= FALSE;
								AspirazioneDX2^.Command^.Aspirazione_OFF := TRUE;
								AspirazioneSX2^.Command^.Aspirazione_ON 	:= FALSE;
								AspirazioneSX2^.Command^.Aspirazione_OFF := TRUE;
								StatoPinza.ElementoPrelevato := FALSE;
								TFTimerSet(ADR(Timeout),3000,TRUE);
								TFCommandCase(ADR(CmdExe),60,CommandCase_JMP);
				
							(* Case 70: Ativazione Tastatori *)
							70:	
								//CilindroTasteggio^.Command.Activation 		:= TRUE;
								//CilindroTasteggio^.Command.Deactivation 	:= FALSE;
								TFTimerSet(ADR(Timeout),3000,TRUE);
								TFCommandCase(ADR(CmdExe),70,CommandCase_JMP);
								
							(* Case 71: Disattivazione Aspirazione SX *)
							71:	
								//CilindroTasteggio^.Command.Activation 		:= FALSE;
								//CilindroTasteggio^.Command.Deactivation 	:= TRUE;
								TFTimerSet(ADR(Timeout),3000,TRUE);
								TFCommandCase(ADR(CmdExe),70,CommandCase_JMP);

							ELSE
								TFError(ErrNOCMDCASE,ErrNULL,ADR(CmdExe),ADR(State),ADR(Error),ADR(ErrorLog));
						END_CASE;

					100:CASE MAN_Cmd OF
							0:	;
							ELSE
								TFError(ErrNOCMDCASE,ErrNULL,ADR(CmdExe),ADR(State),ADR(Error),ADR(ErrorLog));
						END_CASE;

					ELSE
						TFError(ErrNOCMDCASE,ErrNULL,ADR(CmdExe),ADR(State),ADR(Error),ADR(ErrorLog));
				END_CASE;

				//IF CmdExe.CmdCase = 0 THEN
					//TFCommandCase(ADR(CmdExe),1,CommandCase_INC);
				//END_IF

			(* Case 1 - *)
			1: 	IF (MAN_Cmd = 0) OR TFTimerDone(ADR(Timeout)) THEN
					(* Clear All Output Here *)
					;
					TFStateUpdate(ADR(State),StateMAN_END);
					TFCommandExeClear(ADR(CmdExe));
				END_IF;

			
			(* Case 10 - CilindroApertura *)
			10: 
				IF CilindroApertura^.Status.CommandDone THEN
					CilindroApertura^.Command.Activation 	:= FALSE;
					CilindroApertura^.Command.Deactivation 	:= FALSE;
					TFCommandCase(ADR(CmdExe),100,CommandCase_JMP);
				ELSIF CilindroApertura^.Status.ErrorID <> ErrNULL THEN
					TFClearAllCmdModulePinzaCompleta(AspirazioneDX1,AspirazioneSX1,AspirazioneDX2,AspirazioneSX2,CilindroApertura,CilindroSbloccoRotazione,CilindroSbloccoBascolante,AspirazioneFaldaDX,AspirazioneFaldaSX);
					TFError(ErrCYLINDER,CilindroApertura^.Status.ErrorID,ADR(CmdExe),ADR(State),ADR(Error),ADR(ErrorLog));
				END_IF

			(* Case 20 - CilindroSbloccoRotazione *)
			20: 
				IF CilindroSbloccoRotazione^.Status.CommandDone THEN
					CilindroSbloccoRotazione^.Command.Activation 	:= FALSE;
					CilindroSbloccoRotazione^.Command.Deactivation 	:= FALSE;
					TFCommandCase(ADR(CmdExe),100,CommandCase_JMP);
				ELSIF CilindroSbloccoRotazione^.Status.ErrorID <> ErrNULL THEN
					TFClearAllCmdModulePinzaCompleta(AspirazioneDX1,AspirazioneSX1,AspirazioneDX2,AspirazioneSX2,CilindroApertura,CilindroSbloccoRotazione,CilindroSbloccoBascolante,AspirazioneFaldaDX,AspirazioneFaldaSX);
					TFError(ErrCYLINDER,CilindroSbloccoRotazione^.Status.ErrorID,ADR(CmdExe),ADR(State),ADR(Error),ADR(ErrorLog));
				END_IF

			(* Case 30 - AspirazioneFaldaDX *)
			30: 
				IF AspirazioneFaldaDX^.Status.CommandDone THEN
					AspirazioneFaldaDX^.Command.Activation 	:= FALSE;
					AspirazioneFaldaDX^.Command.Deactivation 	:= FALSE;
					TFCommandCase(ADR(CmdExe),100,CommandCase_JMP);
				ELSIF AspirazioneFaldaDX^.Status.ErrorID <> ErrNULL THEN
					TFClearAllCmdModulePinzaCompleta(AspirazioneDX1,AspirazioneSX1,AspirazioneDX2,AspirazioneSX2,CilindroApertura,CilindroSbloccoRotazione,CilindroSbloccoBascolante,AspirazioneFaldaDX,AspirazioneFaldaSX);
					TFError(ErrCYLINDER,AspirazioneFaldaDX^.Status.ErrorID,ADR(CmdExe),ADR(State),ADR(Error),ADR(ErrorLog));
				END_IF

			(* Case 40 - AspirazioneFaldaSX *)
			40: 
				IF AspirazioneFaldaSX^.Status.CommandDone THEN
					AspirazioneFaldaSX^.Command.Activation 	:= FALSE;
					AspirazioneFaldaSX^.Command.Deactivation 	:= FALSE;
					TFCommandCase(ADR(CmdExe),100,CommandCase_JMP);
				ELSIF AspirazioneFaldaSX^.Status.ErrorID <> ErrNULL THEN
					TFClearAllCmdModulePinzaCompleta(AspirazioneDX1,AspirazioneSX1,AspirazioneDX2,AspirazioneSX2,CilindroApertura,CilindroSbloccoRotazione,CilindroSbloccoBascolante,AspirazioneFaldaDX,AspirazioneFaldaSX);
					TFError(ErrCYLINDER,AspirazioneFaldaSX^.Status.ErrorID,ADR(CmdExe),ADR(State),ADR(Error),ADR(ErrorLog));
				END_IF

			(* Case 50 - AspirazioneSX *)
			50: 
				IF AspirazioneSX1^.Status.CommandDone AND AspirazioneDX1^.Status.CommandDone AND
					AspirazioneSX2^.Status.CommandDone AND AspirazioneDX2^.Status.CommandDone THEN
						AspirazioneDX1^.Command^.Aspirazione_ON 	:= FALSE;
						AspirazioneDX1^.Command^.Aspirazione_OFF	:= FALSE;
						AspirazioneSX1^.Command^.Aspirazione_ON 	:= FALSE;
						AspirazioneSX1^.Command^.Aspirazione_OFF	:= FALSE;
						AspirazioneDX2^.Command^.Aspirazione_ON 	:= FALSE;
						AspirazioneDX2^.Command^.Aspirazione_OFF	:= FALSE;
						AspirazioneSX2^.Command^.Aspirazione_ON 	:= FALSE;
						AspirazioneSX2^.Command^.Aspirazione_OFF	:= FALSE;
						TFCommandCase(ADR(CmdExe),100,CommandCase_JMP);
				ELSIF AspirazioneSX1^.Status.ErrorID <> ErrNULL THEN
					TFClearAllCmdModulePinzaCompleta(AspirazioneDX1,AspirazioneSX1,AspirazioneDX2,AspirazioneSX2,CilindroApertura,CilindroSbloccoRotazione,CilindroSbloccoBascolante,AspirazioneFaldaDX,AspirazioneFaldaSX);
					TFError(ErrCYLINDER,AspirazioneSX1^.Status.ErrorID,ADR(CmdExe),ADR(State),ADR(Error),ADR(ErrorLog));
				ELSIF AspirazioneDX1^.Status.ErrorID <> ErrNULL THEN
					TFClearAllCmdModulePinzaCompleta(AspirazioneDX1,AspirazioneSX1,AspirazioneDX2,AspirazioneSX2,CilindroApertura,CilindroSbloccoRotazione,CilindroSbloccoBascolante,AspirazioneFaldaDX,AspirazioneFaldaSX);
					TFError(ErrCYLINDER,AspirazioneDX1^.Status.ErrorID,ADR(CmdExe),ADR(State),ADR(Error),ADR(ErrorLog));
				END_IF

